// init controller
FOR i:=1 TO 3 DO
	currentRatioMotor2Jnt:=GVL_system_parameters.arm_joint_transmition_efficiency[i-1+Gvl_IO.Joint6]*GVL_system_parameters.arm_joint_torque_constant[i-1+Gvl_IO.Joint6]
							*GVL_system_parameters.transmission_ratio[m_armIdx, i-1+Gvl_IO.Joint6]/1000;
	m_jntPIDCtrl[i].init(GVL_system_parameters.cycle_robot,m_macroJntKp[i],m_macroJntKd[i],m_macroJntKi[i],
		m_macroJntKiLimit[i]* currentRatioMotor2Jnt,	m_macroJnttrlLimit[i]*currentRatioMotor2Jnt);
END_FOR

// init low pass filter
FOR i:=1 TO 3 DO
	m_cmdPosLpf[i].init(i_filterOrd:=1,i_cutoffFreq:=m_jntTargetPosLpfCutoffFreq,i_sampleFreq:=1000);
	m_curJntVelLpf[i].init(i_filterOrd:=1,i_cutoffFreq:=m_curJntVelLpfCutoffFreq,i_sampleFreq:=1000);
END_FOR
END_METHOD

METHOD run : BOOL
VAR_INPUT
	// target joint position in DH model 3
	i_targetJntPos:ARRAY[1..3] OF LREAL;

END_VAR

VAR_OUTPUT
	// motor control current
	o_cmdMotorTrq:ARRAY[1..3] OF LREAL;
END_VAR

VAR
	i: INT;
END_VAR
// fitl target joint position
FOR i:=1 TO 3 DO
	m_targetJntPos[i]:=m_cmdPosLpf[i].run(i_targetJntPos[i]);
END_FOR

// get current joint position
m_curJntPos[1]:=Robot_Status.Robot_Current_DH_Joint_Position_M3[m_armIdx].q1;
m_curJntPos[2]:=Robot_Status.Robot_Current_DH_Joint_Position_M3[m_armIdx].q2;
m_curJntPos[3]:=Robot_Status.Robot_Current_DH_Joint_Position_M3[m_armIdx].q3;

// get current joint velocity
m_curJntVel[1]:=m_curJntVelLpf[1].run(Robot_Status.Robot_Current_Joint_Velocity_V2[m_armIdx,6]);
m_curJntVel[2]:=m_curJntVelLpf[2].run(Robot_Status.Robot_Current_Joint_Velocity_V2[m_armIdx,10]);
m_curJntVel[3]:=m_curJntVelLpf[3].run(Robot_Status.Robot_Current_Joint_Velocity_V2[m_armIdx,11]);

// interpolate command position
FOR i:=1 TO 3 DO
	m_cmdJntVel[i]:=LIMIT(-m_maxJntVel[i],(m_targetJntPos[i]-m_cmdJntPos[i])/GVL_system_parameters.cycle_robot, m_maxJntVel[i]);
	m_cmdJntPos[i]:=m_cmdJntPos[i]+m_cmdJntVel[i]*GVL_system_parameters.cycle_robot;
END_FOR  

// joint position control torque control
FOR i:=1 TO 3 DO
	o_cmdMotorTrq[i]:=0;
	m_posErr[i]:=m_cmdJntPos[i]-m_curJntPos[i];
	m_cmdJntTrq[i]:=m_jntPIDCtrl[i].run(m_cmdJntPos[i],m_curJntPos[i], m_cmdJntVel[i], m_curJntVel[i]);
END_FOR

// safety check
FOR i:=1 TO 3 DO
	IF ABS(m_posErr[i])>m_safetyPosErr[i] THEN
		run := FALSE;
		RETURN;
	END_IF
END_FOR

// motor control current
o_cmdMotorTrq[1]:=gvl_system_parameters.Joint_Motion_direction[m_armIdx,6]*(m_cmdJntTrq[1]+Robot_Status.Robot_Joint_Gravity[1].q6);
o_cmdMotorTrq[2]:=gvl_system_parameters.Joint_Motion_direction[m_armIdx,10]*(m_cmdJntTrq[2]+Robot_Status.Robot_Joint_Gravity[1].q10);
o_cmdMotorTrq[3]:=gvl_system_parameters.Joint_Motion_direction[m_armIdx,11]*(m_cmdJntTrq[3]+Robot_Status.Robot_Joint_Gravity[1].q11);
run := TRUE;
END_METHOD

END_FUNCTION_BLOCK

// ---- FBs_CartControlles/FB_CartPinDeploy.TcPOU
FUNCTION_BLOCK FB_CartPinDeploy EXTENDS FB_CartCtrlBase
VAR_INPUT
END_VAR
VAR_OUTPUT
END_VAR
VAR

	m_actJntPos: Vec8d;
	m_tarJntPos: Vec8d;
	m_initJntPos : Vec8d;
	m_tarJntInc : Vec8d;
	m_maxJntCurrent : ARRAY [1..2] OF LREAL := [1000,1000];
	m_pinDeployed : ARRAY [1..2] OF BOOL; 
	
	m_carJntSoftwareLimit :ARRAY [1..2] OF LREAL := [0.005, 2*g_deg2Rad, 0.005, 2*g_deg2Rad];
	
	// time threshold to 5-8joint after it's enabled
	m_cartAdjustStartWaitTime :LREAL := 0.2;
	
	//adjust start  time 
	m_adjustStartTime :LREAL;

	m_jntOTG :ARRAY [1..2] OF FB_secOrdTrajFilter;
END_VAR

// override this function in each exact controller
METHOD PROTECTED calcCmdJntPos : BOOL
VAR_IN_OUT CONSTANT
	// slave cart joint data
	i_slaveCart :FB_SlaveCart;
END_VAR

VAR
	i:INT;
END_VAR
//In this method, 8 represents the overhang angle
m_adjustStartTime :=LIMIT(0, m_adjustStartTime + g_cartCtrlCycleTime, 1);
m_actJntPos := i_slaveCart.curJntPos;
IF m_adjustStartTime > m_cartAdjustStartWaitTime THEN
	FOR i:=1 TO 2 DO
		IF ABS(i_slaveCart.curJntCurrent[i]) > m_maxJntCurrent[i] THEN
			m_pinDeployed[i] := TRUE;
			m_tarJntPos[i] := m_actJntPos[i];
		END_IF
		
		IF FALSE = m_pinDeployed[i] THEN
			m_tarJntPos[i] := m_actJntPos[i] + GVL_CartControlParameters.g_maxJntVel[i] * g_cartCtrlCycleTime;
		END_IF
		m_jntOTG[i].run(i_targetPos:= m_tarJntPos[i], i_targetVel:= 0.0, o_cmdAcc=> , o_cmdVel=> , o_cmdPos=>m_cmdJntPos[i] );
	END_FOR
	
	IF m_pinDeployed[1] AND m_pinDeployed[2] THEN
		m_isFinished := TRUE;
	END_IF

END_IF
END_METHOD

// override this function in each exact controller
// NOTICE: set joint control mode here, and do some initialization if needed
METHOD PUBLIC init : BOOL
VAR_IN_OUT CONSTANT
	i_slaveCart	:FB_SlaveCart;
END_VAR
VAR_IN_OUT 
	r_cartCtrlCmd :ST_SlaveArmCtrlCmds;
END_VAR
VAR
	i:INT;
END_VAR
//m_holdLastCmds := checkToHoldLastCmds(i_slaveCart);
m_holdLastCmds := checkToHoldLastCmds(i_slaveCart);

SUPER^.init(i_slaveCart,r_cartCtrlCmd);

m_jntEnableFlag[1] :=1;
m_jntEnableFlag[2] :=1;

m_jntOPMode[1]:= DriverOPMode_Pos;
m_jntOPMode[2]:= DriverOPMode_Pos;

m_pinDeployed[1] := FALSE;
m_pinDeployed[2] := FALSE;

m_jntOTG[1].init(i_curCmdPos:= m_cmdJntPos[1], i_curCmdVel:= 0, i_maxV:=GVL_CartControlParameters.g_maxJntVel[1] , i_maxA:=GVL_CartControlParameters.g_maxJntAcc[1] , i_Ts:=g_cartCtrlCycleTime );
m_jntOTG[2].init(i_curCmdPos:= m_cmdJntPos[2], i_curCmdVel:= 0, i_maxV:=GVL_CartControlParameters.g_maxJntVel[2] , i_maxA:=GVL_CartControlParameters.g_maxJntAcc[2] , i_Ts:=g_cartCtrlCycleTime );

m_adjustStartTime := 0;
// update commands to arm
copyCmds(r_cartCtrlCmd);
END_METHOD

END_FUNCTION_BLOCK

// ---- FBs_RobotDynamics/FB_FullArmKinematic.TcPOU
FUNCTION_BLOCK FB_FullArmKinematic
VAR
	m_armIdx :INT :=1;
	
	// nominal DH parameters
	//% setup arm
//% 1        0      0   q1      0
//% 2        90     a2   0      q2
//% 3        -90     0   0       q3
//% 4        0       0   q4      d4
//% 5        -90      0   q5      0

//% paramters definiton:
//% a: distance from joint5 to joint 6 on tool
//% b: distantce form joint 6 to tcp on tool
//% DH definition:
//% index    alpha   a        theta           d
//% 1        90      0        J1+180          0
//% 2        90     42.45     J2-61.935       0
//% P1       0      254       -J2-200.065     0
//% P2       0      305       J2+82              0
//% 3        -90     119.5    0               J3-224.133
//% 4        0       0        J4              -L
//% 5        90      0        J5              0
//% 6        90      a        J6              0
//% tcp      0       b        0               0
	m_armNominalDH :ARRAY[1..14] OF Vec4d;
	
	// calibrated DH parameters err
//	% setupDHErr=[   0   0   dq1     0;
//%                0  da2   0      dq2;
//%                0  0   0       dq3;
//%                0  0   dq4      0;
//%                0  da5  dq5      0];
//% slaveDHErr=[  0       0           dq6      0;
//%               0      0            dq7      da7;
//%               0      0            dq8       0;
//%               0     0               dq9       0;
//%               0     0           0          dq10;
//%                 0       0          0      0];
// m_DHErr=[dq1,da2,dq2, dq3, dq4, da5, dq5,  dq6, dq7, da7, dq8, dq9, dq10]
	m_DHErr:ARRAY[1..13] OF LREAL := [13(0.0)];
	
	// hanger base matrix
	m_baseRadiu :LREAL :=0.17;
	m_baseAng:LREAL := 60.0*g_deg2rad;
	m_baseFrame :ST_Frame;
	
	m_currentDH :ARRAY[1..14] OF Vec4d;
	
	m_tcpFrame :ST_Frame;
	
	m_useCaliData :BOOL:=true;
END_VAR

METHOD init : BOOL
VAR_INPUT
	i_armIdx:INT;
END_VAR
VAR 
	i,j:INT;
END_VAR
m_armIdx := i_armIdx;

FOR i:=1 TO 5 DO 
	FOR j:=1 TO 4 DO
		m_armNominalDH[i][j]:= GVL_SetupArmKinematic.g_setupArmDH[i,j];
	END_FOR	
END_FOR
m_armNominalDH[2][2]:=GVL_SetupArmKinematic.g_setupA2[m_armIdx];
m_armNominalDH[4][4]:=GVL_SetupArmKinematic.g_setupD4[m_armIdx];

FOR i:=1 TO 9 DO 
	FOR j:=1 TO 4 DO
		m_armNominalDH[i+5][j]:= GVL_SlaveArmKinematic.g_slaveArmFullDH[i,j];
	END_FOR	
END_FOR


FOR i:=1 TO 13 DO
	IF m_useCaliData THEN
		m_DHErr[i] := GVL_SlaveArmKinematic.g_slaveArmDHErr[m_armIdx, i];
	ELSE
		m_DHErr[i]:=0;
	END_IF
END_FOR



m_armNominalDH[1][3]:=m_armNominalDH[1][3]+m_DHErr[1];
m_armNominalDH[2][2]:=m_armNominalDH[2][2]+m_DHErr[2];
m_armNominalDH[2][4]:=m_armNominalDH[2][4]+m_DHErr[3];
m_armNominalDH[3][4]:=m_armNominalDH[3][4]+m_DHErr[4];
m_armNominalDH[4][3]:=m_armNominalDH[4][3]+m_DHErr[5];
m_armNominalDH[5][2]:=m_armNominalDH[5][2]+m_DHErr[6];
m_armNominalDH[5][3]:=m_armNominalDH[5][3]+m_DHErr[7];

m_armNominalDH[6][3]:=m_armNominalDH[6][3]+m_DHErr[8];
m_armNominalDH[7][3]:=m_armNominalDH[7][3]+m_DHErr[9];
m_armNominalDH[7][4]:=m_armNominalDH[7][4]+m_DHErr[10];
m_armNominalDH[8][3]:=m_armNominalDH[8][3]+m_DHErr[11];
m_armNominalDH[9][3]:=m_armNominalDH[9][3]+m_DHErr[12];
m_armNominalDH[10][4]:=m_armNominalDH[10][4]+m_DHErr[13];

m_baseFrame.m_pos[3]:=0;
IF (m_armIdx=1) THEN
	m_baseFrame.m_pos[1]:=-m_baseRadiu; 
	m_baseFrame.m_pos[2]:=0;
	
ELSIF (m_armIdx=2) THEN
	m_baseFrame.m_pos[1]:=-m_baseRadiu*COS(m_baseAng); 
	m_baseFrame.m_pos[2]:=-m_baseRadiu*SIN(m_baseAng);
	
ELSIF (m_armIdx=3) THEN	
	m_baseFrame.m_pos[1]:=m_baseRadiu*COS(m_baseAng); 
	m_baseFrame.m_pos[2]:=-m_baseRadiu*SIN(m_baseAng); 
	
ELSIF (m_armIdx=4) THEN	
	m_baseFrame.m_pos[1]:=m_baseRadiu; 
	m_baseFrame.m_pos[2]:=0;
END_IF

IF m_useCaliData THEN
	m_baseFrame.m_pos[1]:=m_baseFrame.m_pos[1]+GVL_SlaveArmKinematic.g_slaveArmBaseErr[m_armIdx,1];
	m_baseFrame.m_pos[2]:=m_baseFrame.m_pos[2]+GVL_SlaveArmKinematic.g_slaveArmBaseErr[m_armIdx,2];
END_IF
m_baseFrame.m_rot[1,1]:=0;
m_baseFrame.m_rot[2,1]:=1;
m_baseFrame.m_rot[3,1]:=0;

m_baseFrame.m_rot[1,2]:=-1;
m_baseFrame.m_rot[2,2]:=0;
m_baseFrame.m_rot[3,2]:=0;

m_baseFrame.m_rot[1,3]:=0;
m_baseFrame.m_rot[2,3]:=0;
m_baseFrame.m_rot[3,3]:=1;
END_METHOD

METHOD run : BOOL
VAR_IN_OUT CONSTANT
	// setup joint angle
	i_setupPos : vec5d;
	
	// slave DH joint angle
	i_slaveDHJntPos :Vec6d;
	
	// instrument
	i_instruStatus :ST_InstruStatus;
END_VAR
VAR_IN_OUT
	r_tcpPose:ST_Frame;
END_VAR
VAR
	i:INT;
	T1,T2 :ST_Frame;
END_VAR
// instrument parameters
m_armNominalDH[11][4]:=-GVL_SlaveArmKinematic.g_L;
m_armNominalDH[13][2]:=GVL_SlaveArmKinematic.g_a;
m_armNominalDH[14][2]:=GVL_SlaveArmKinematic.g_b;
FOR i:=1 TO g_instruTypeNum DO 
	IF g_instruTypePool[i].m_InstruID = i_instruStatus.m_type THEN
		m_armNominalDH[11][4]:=-(g_instruTypePool[i].m_rodLength-GVL_SlaveArmKinematic.g_panelHeight);
		m_armNominalDH[13][2]:=g_instruTypePool[i].m_headLength;
		m_armNominalDH[14][2]:=g_instruTypePool[i].m_fingerLength;
		EXIT;
	END_IF
END_FOR

// add joint position
m_currentDH:=m_armNominalDH;
m_currentDH[1][3]:=m_currentDH[1][3]+i_setupPos[1];
m_currentDH[2][4]:=m_currentDH[2][4]+i_setupPos[2];
m_currentDH[3][4]:=m_currentDH[3][4]+i_setupPos[3];
m_currentDH[4][3]:=m_currentDH[4][3]+i_setupPos[4];
m_currentDH[5][3]:=m_currentDH[5][3]+i_setupPos[5];
m_currentDH[6][3]:=m_currentDH[6][3]+i_slaveDHJntPos[1];
m_currentDH[7][3]:=m_currentDH[7][3]+i_slaveDHJntPos[2];
m_currentDH[8][3]:=m_currentDH[8][3]-i_slaveDHJntPos[2];
m_currentDH[9][3]:=m_currentDH[9][3]+i_slaveDHJntPos[2];
m_currentDH[10][4]:=m_currentDH[10][4]+i_slaveDHJntPos[3];
m_currentDH[11][3]:=m_currentDH[11][3]+i_slaveDHJntPos[4];
m_currentDH[12][3]:=m_currentDH[12][3]+i_slaveDHJntPos[5];
m_currentDH[13][3]:=m_currentDH[13][3]+i_slaveDHJntPos[6];

m_tcpFrame:= m_baseFrame;
FOR i:=1 TO 14 DO 
	T1:=DHTrans(m_currentDH[i]);
	T2:=transform(m_tcpFrame,T1);
	m_tcpFrame:=T2;
END_FOR
matMultiply(T2.m_rot, GVL_SlaveArmKinematic.g_tcpRotation, m_tcpFrame.m_rot);

r_tcpPose:=m_tcpFrame;
END_METHOD

END_FUNCTION_BLOCK

// ---- FBs_RobotDynamics/FB_InstruViewCheck.TcPOU
FUNCTION_BLOCK FB_InstruViewCheck
VAR
	
	// scoep projection matrix 
	//SN: HA21938730
	m_scopeRot :Mat3d :=[0.9983, -0.0327, 0.048, 
						0.0319, 0.9993, 0.0179,
						-0.0486, -0.0164, 0.9987];
	m_scopePos :Vec3d:= [0.005, 0.000214, 0.00386];
	m_scopeFocal :LREAL :=1400;
	
//	//SN: HA20160831
//	m_scopeRot :Mat3d :=[0.9952, 0.0185, 0.0961, 
//						-0.0177, 0.9998, -0.0099,
//						-0.0963, 0.0081, 0.9953];
//	m_scopePos :Vec3d:= [-0.0006967, 0.001848, -0.005];
//	m_scopeFocal :LREAL :=1420;

	// arm kinematic function block
	m_armKinematic :ARRAY[1..g_sArmNum] OF FB_FullArmKinematic;
	
	// instrument pose
	m_instruReady:ARRAY[1..g_sArmNum] OF BOOL;
	m_instruPose :ARRAY[1..g_sArmNum] OF ST_Frame;
	
	// endoscope pose
	m_scopeReady :BOOL;
	m_scopePose : ST_Frame;
	
	// instrument pose in scope 
	m_instruPoseInScope :ARRAY[1..g_sArmNum] OF ST_Frame;
	
	// instrument position in image([x_pixel, y_pixel, z_dir])
	m_instruImgPos :ARRAY[1..g_sArmNum] OF Vec3d;
	
	// out-view instrument position on image boundary([x_pixel, y_pixel, z_dir])
	 m_instruImgBoundPos :ARRAY[1..g_sArmNum] OF Vec3i;
	 
	 // image boundary
	 m_imgWidth :INT := 960;
	 m_ImgHeight :INT :=540;
	
END_VAR

METHOD init : BOOL
VAR_INPUT
END_VAR
VAR
	i:INT;
END_VAR
FOR i:=1 TO g_sArmNum DO
	m_instruReady[i]:=FALSE;
	m_armKinematic[i].init(i);
	m_instruImgPos[i]:=g_zeroVec3d;
	m_instruImgBoundPos[i]:=g_zeroVec3i;
END_FOR
m_scopeReady:=FALSE;
END_METHOD

METHOD run : BOOL
VAR_IN_OUT CONSTANT
	// setup joint position
	i_setupJntPos :ARRAY[1..g_sArmNum] OF Vec5d;
	
	// slave joint position
	i_slaveDHJntPos :ARRAY[1..g_sArmNum] OF Vec6d;
	
	// instrument info
	i_instruInfo : ARRAY[1..g_sArmNum] OF ST_InstruStatus;
END_VAR

VAR
	i:INT;
	tmpFrame: ST_Frame;
	newPos:Vec3d ;
	xb,yb : INT;
END_VAR
m_scopeReady := FALSE;
// update instrument and endoscope pose
FOR i:=1 TO g_sArmNum DO 
	m_instruReady[i]:=FALSE;
	IF i_instruInfo[i].m_ready THEN
		m_instruReady[i]:=TRUE;
		m_armKinematic[i].run(i_setupJntPos[i],i_slaveDHJntPos[i], i_instruInfo[i], m_instruPose[i]);
		IF i_instruInfo[i].m_type = InstruType_Endoscope THEN
			m_scopePose := m_instruPose[i];
			m_scopeReady := TRUE;
		END_IF
	END_IF
	
	m_instruImgPos[i]:=g_zeroVec3d;
	m_instruImgBoundPos[i]:=g_zeroVec3i;
END_FOR

IF m_scopeReady THEN
	FOR i:=1 TO g_sArmNum DO
		IF m_instruReady[i] THEN
			// calculate instrument pose in endoscope
			tmpFrame :=invFrame(m_scopePose);
			m_instruPoseInScope[i] := transform(tmpFrame, m_instruPose[i]);
			
			// calculate instrument in image
			IF ABS(m_instruPoseInScope[i].m_pos[3])>0.02 THEN
				MatMultiVec(m_scopeRot, m_instruPoseInScope[i].m_pos, newPos);
				vecSelfAdd(newPos, m_scopePos);
				m_instruImgPos[i][1]:= m_scopeFocal* newPos[1]/ABS(newPos[3]);
				m_instruImgPos[i][2]:= -m_scopeFocal * newPos[2]/ABS(newPos[3]);
				m_instruImgPos[i][3] := sign(newPos[3]); 
			END_IF
			
			// check if instrument is  out of view
			IF ABS(m_instruImgPos[i][1])>m_imgWidth OR ABS(m_instruImgPos[i][2])>m_ImgHeight THEN
				IF ABS(m_instruImgPos[i][2]/m_instruImgPos[i][1]) > INT_TO_LREAL( m_ImgHeight)/INT_TO_LREAL(m_imgWidth) THEN
					yb:=sign(m_instruImgPos[i][2])*m_ImgHeight;
					xb:=LREAL_TO_INT(m_instruImgPos[i][1]*yb/m_instruImgPos[i][2]);
				ELSE
					xb:=sign(m_instruImgPos[i][1])*m_imgWidth;
					yb:=LREAL_TO_INT(m_instruImgPos[i][2]*xb/m_instruImgPos[i][1]);
				END_IF
				m_instruImgBoundPos[i][1]:=xb;
				m_instruImgBoundPos[i][2]:=yb;
				m_instruImgBoundPos[i][3]:=LREAL_TO_INT(m_instruImgPos[i][3]);
			END_IF
						
		END_IF
	END_FOR
END_IF
END_METHOD

END_FUNCTION_BLOCK

// ---- FBs_RobotDynamics/FB_SlaveDynamic.TcPOU
FUNCTION_BLOCK FB_SlaveDynamic
VAR_INPUT
END_VAR
VAR_OUTPUT
END_VAR
VAR CONSTANT
	//kinematic constraint
	//  q3 =- q2;           
	//  q4 = q2;             
 	// jacobian with active joints
 	// jaco_DH*qdot_DH = jaco_DH * (A * qdot_active)= jaco * qdot_active
 	// q_DH=[q1,q2,q3,q4,q5];
 	// q_active=[q1,q2,q5]
	m_jacoA :Mat53 :=
	[   1,  0,  0,
        0,  1,  0,
		0, -1,  0,
		0,  1,  0,
		0,  0,  1];
	
	// DH parameters for dynamic model
	(*slaveDH=[   deg90       0           q1+pi                502.591/1000;
            deg90       42.45/1000  q2-deg2rad(61.935)   0;
            0           254/1000    q3-deg2rad(200.065) 0;
            0           305/1000    q4+deg2rad(82)       0;
            -deg90      119.5/1000  0                           q5-224.133/1000];*)
	m_armOriginalDH:ARRAY[1..5,1..4] OF LREAL :=
	[PI/2,       0,         	   pi,     502.591/1000,          
	PI/2,       42.45/1000,  	-61.935*g_deg2rad,  0, 		
	0,           254.0/1000,  	-200.065*g_deg2rad, 0,  
	0,           305.0/1000,    	82*g_deg2rad,      	0, 			
	-PI/2,      119.5/1000,   0,	-224.133/1000];
	
END_VAR

VAR
			
	m_armIdx :INT;
	m_armDH:ARRAY[1..5] OF Vec4d;
	
	// dynamic parameters
	m_linkMass :ARRAY[1..5] OF LREAL;
	m_linkCOM :ARRAY[1..5] OF Vec3d;
	m_linkInertia :ARRAY[1..5] OF Mat3d;
		
	// frame of each joint
	m_jntFrame :ARRAY[1..5] OF ST_Frame;
	
	// jacobian of mass center
	m_Jp :ARRAY[1..5] OF Mat3d;
	m_Jo :ARRAY[1..5] OF Mat3d;
	
	// motor inertia at link size
	m_motorInertia :Vec3d;
	
	// mass matrix in joint space
	m_massMat :Mat3d;
	
END_VAR

METHOD init : BOOL
VAR_INPUT
	i_armIdx :INT ;
END_VAR

VAR
	i,j:INT;
END_VAR
m_armIdx:=i_armIdx;

m_linkMass:=GVL_SlaveArmDynamics.g_linkMass;
FOR i:=1 TO 5 DO
	m_linkCOM[i][1]:=GVL_SlaveArmDynamics.g_linkCOM[i,1];
	m_linkCOM[i][2]:=GVL_SlaveArmDynamics.g_linkCOM[i,2];
	m_linkCOM[i][3]:=GVL_SlaveArmDynamics.g_linkCOM[i,3];
	
	m_linkInertia[i][1,1]:=GVL_SlaveArmDynamics.g_linkInertia[i,1];
	m_linkInertia[i][2,2]:=GVL_SlaveArmDynamics.g_linkInertia[i,2];
	m_linkInertia[i][3,3]:=GVL_SlaveArmDynamics.g_linkInertia[i,3];
	m_linkInertia[i][1,2]:=GVL_SlaveArmDynamics.g_linkInertia[i,4];
	m_linkInertia[i][1,3]:=GVL_SlaveArmDynamics.g_linkInertia[i,5];
	m_linkInertia[i][2,3]:=GVL_SlaveArmDynamics.g_linkInertia[i,6];
	m_linkInertia[i][2,1]:=m_linkInertia[i][1,2];
	m_linkInertia[i][3,1]:=m_linkInertia[i][1,3];
	m_linkInertia[i][3,2]:=m_linkInertia[i][2,3];
END_FOR

FOR i:=1 TO 3 DO
	m_motorInertia[i]:=GVL_SlaveArmDynamics.g_motorInertia[i]*GVL_SlaveMotorParameters.g_motorReduction[i]*GVL_SlaveMotorParameters.g_motorReduction[i];
END_FOR

FOR i:=1 TO 5 DO
	FOR j:=1 TO 4 DO 
		m_armDH[i][j] := m_armOriginalDH[i,j];
	END_FOR
END_FOR
END_METHOD

PROPERTY PUBLIC jntMassMat : Mat3d
GET
jntMassMat := m_massMat;
END_GET
END_PROPERTY

// update dynamic and kinematic data 
METHOD updateDynamic : BOOL
VAR_IN_OUT CONSTANT
	i_jntPos : Vec8d;
END_VAR
VAR
	tmpJntPos :Vec8d;
	
	i,j:INT;
	m,n :INT;
	linkMassMat :ARRAY[1..5] OF Mat3d;
	linkInerMat :ARRAY[1..5] OF Mat3d;
	inertia,Rt :Mat3d;
	
	JotI,Jot, Jpt :Mat3d;
	
	tmpMat3d :Mat3d;

	
END_VAR
// update kinematic 
updateKinematic(i_jntPos);

// joint space mass matrix
// massMat=m*Jp'*Jp+Jo'*R*I*R'*Jo
FOR i:=1 TO 5 DO
	// iner=R*I*R'
	matMultiply(m_jntFrame[i].m_rot,m_linkInertia[i],tmpMat3d);
	matTranspose(m_jntFrame[i].m_rot, Rt);
	matMultiply(tmpMat3d,Rt,inertia);
	
	// m*Jp'*Jp+Jo'*iner*Jo
	matTranspose(m_Jp[i],Jpt);
	matMultiply(Jpt,m_Jp[i], tmpMat3d);
	matMultiNum(tmpMat3d, m_linkMass[i],linkMassMat[i]);
	
	matTranspose(m_Jo[i],Jot);
	matMultiply(Jot,inertia, JotI);
	matMultiply(JotI,m_Jo[i],linkInerMat[i]);
END_FOR

// total mass mat
m_massMat :=g_zeroMat3d;
FOR i:=1 TO 5 DO
	matSelfAdd(m_massMat,linkMassMat[i]);
	matSelfAdd(m_massMat,linkInerMat[i]);
END_FOR

// add motor inertial 
FOR i:=1 TO 3 DO
	m_massMat[i,i]:=m_massMat[i,i]+m_motorInertia[i];
END_FOR
END_METHOD

// only update kinematic data
METHOD PROTECTED updateKinematic : BOOL
VAR_IN_OUT CONSTANT
	i_jntPos : Vec8d;
END_VAR
VAR
	Jp :Mat35;
	Jo :Mat35;
	T :ST_Frame;
	i,j:INT;
	Pc,z,p:Vec3d;
	m,n :INT;
	
END_VAR
// tranform a joint positon to DH ones
m_armDH[1][3] := m_armOriginalDH[1,3] + i_jntPos[1];
m_armDH[2][3] := m_armOriginalDH[2,3] + i_jntPos[2];
m_armDH[3][3] := m_armOriginalDH[3,3] - i_jntPos[2];
m_armDH[4][3] := m_armOriginalDH[4,3] + i_jntPos[2];
m_armDH[5][4] := m_armOriginalDH[5,4] + i_jntPos[3];

// compute joint frame
m_jntFrame[1]:=DHTrans(m_armDH[1]);
T:=DHTrans(m_armDH[2]);
m_jntFrame[2]:=transform(m_jntFrame[1],T);
T:=DHTrans(m_armDH[3]);
m_jntFrame[3]:=transform(m_jntFrame[2],T);
T:=DHTrans(m_armDH[4]);
m_jntFrame[4]:=transform(m_jntFrame[3],T);
T:=DHTrans(m_armDH[5]);
m_jntFrame[5]:=transform(m_jntFrame[4],T);


// jacobian of mass center
FOR i:=1 TO 5 DO 
	Jp := g_zeroMat35;
	Jo := g_zeroMat35;
    T:=m_jntFrame[i];
	// mass center world position
    matMultiVec(T.m_rot,m_linkCOM[i], Pc);
	vecSelfAdd(Pc, T.m_pos);
    FOR j:=1 TO i DO
        T:=m_jntFrame[j];
		z[1]:=T.m_rot[1,3];
		z[2]:=T.m_rot[2,3];
		z[3]:=T.m_rot[3,3];
		IF (5=j) THEN
			Jp[1,j]:=z[1];
			Jp[2,j]:=z[2];
			Jp[3,j]:=z[3];
			Jo[1,j]:=0;
			Jo[2,j]:=0;
			Jo[3,j]:=0;
		ELSE
			vecSub(Pc,T.m_pos,p);
			p:=cross(z,p);
			Jp[1,j]:=p[1];
			Jp[2,j]:=p[2];
			Jp[3,j]:=p[3];
			Jo[1,j]:=z[1];
			Jo[2,j]:=z[2];
			Jo[3,j]:=z[3];			
        END_IF
    END_FOR
	// multiply m_jacoA
	matMultiply(Jp, m_jacoA, m_Jp[i]);
	matMultiply(Jo, m_jacoA, m_Jo[i]);
END_FOR
END_METHOD

END_FUNCTION_BLOCK

// ---- FBs_RobotDynamics/FB_SlaveGravity.TcPOU
FUNCTION_BLOCK FB_SlaveGravity
VAR_INPUT
END_VAR
VAR
	m_armIdx :INT ;

	// current arm parameters
	m_armParams :ARRAY[1..5] OF LREAL;

END_VAR

METHOD getRegMat : BOOL
VAR_INPUT
	// joint position of setup joint, joint6-8
	setupAng :LREAL;
	q1: LREAL;
	q2: LREAL;
	q3: LREAL;
END_VAR

VAR
	s0,c0, s1,c1,s2, c2,d3 :LREAL;
END_VAR

VAR_OUTPUT
	o_regMat:ARRAY[1..3,1..5] OF LREAL;
END_VAR
s0:=SIN(setupAng);
c0:=COS(setupAng);
s1:=SIN(q1);
c1:=COS(q1);
s2:=SIN(q2);
c2:=COS(q2);
d3:=q3;

// joint1
o_regMat[1,1] :=s0*s1*s2*d3;
o_regMat[1,2] :=  s0*s1;
o_regMat[1,3] := -s0*c1;
o_regMat[1,4] := s0*s1*s2;
o_regMat[1,5] := s0*c2*s1 ;

// joint2 
o_regMat[2,1] :=  - (c0*s2*d3+s0*c1*c2*d3);
o_regMat[2,2] := 0;
o_regMat[2,3] := 0;
o_regMat[2,4] :=  - (c0*s2+s0*c1*c2);
o_regMat[2,5] := s0*c1*s2- c0*c2;

// joint3
o_regMat[3,1] :=c0*c2 - s0*c1*s2;
o_regMat[3,2] :=0;
o_regMat[3,3] :=0;
o_regMat[3,4] :=0;
o_regMat[3,5] :=0;
END_METHOD

METHOD init : BOOL
VAR_INPUT
	i_armIdx :INT;
END_VAR
m_armIdx :=i_armIdx;
END_METHOD

METHOD run : Vec3d
VAR_IN_OUT CONSTANT
	// setup joint5 angle
	i_setupPos :LREAL;
	
	// slave joint angle
	i_slaveJntPos :Vec8d;
	
	// instrument
	i_instruStatus :ST_InstruStatus;
END_VAR
VAR
	q1, q2, q3 :LREAL;
	i,j:INT;
	
	// gravity regression matrix
	regMat:ARRAY[1..3,1..5] OF LREAL;
END_VAR
q1 :=LIMIT (GVL_SlaveMotorParameters.g_minJntPos[1], i_slaveJntPos[1], GVL_SlaveMotorParameters.g_maxJntPos[1]);
q2 := LIMIT (GVL_SlaveMotorParameters.g_minJntPos[2], i_slaveJntPos[2], GVL_SlaveMotorParameters.g_maxJntPos[2]);
q3 := LIMIT (GVL_SlaveMotorParameters.g_minJntPos[3], i_slaveJntPos[3], GVL_SlaveMotorParameters.g_maxJntPos[3]);


// get regression matrx
getRegMat(i_setupPos, q1, q2, q3, o_regMat=>regMat);

// determine current arm parameters
IF FALSE = i_instruStatus.m_ready THEN
	// arm only
	FOR i:=1 TO 5 DO
		m_armParams[i]:=GVL_SlaveArmDynamics.g_gravityParam[m_armIdx,i];
	END_FOR

// endoscope
ELSIF InstruType_endoscope = i_instruStatus.m_type THEN 
	FOR i:=1 TO 5 DO
		m_armParams[i]:=GVL_SlaveArmDynamics.g_gravityParam[m_armIdx,i]+GVL_SlaveArmDynamics.g_gravityEndoscope[i];
	END_FOR

// instrument
ELSE
	FOR i:=1 TO 5 DO
		m_armParams[i]:=GVL_SlaveArmDynamics.g_gravityParam[m_armIdx,i]+GVL_SlaveArmDynamics.g_gravityInstrument[i];
	END_FOR
// TODO:Trocar
END_IF

// calculate gravity torque
FOR i:=1 TO 3 DO
	run[i]:=0;
	FOR j:=1 TO 5 DO
		run[i]:=run[i]+regMat[i,j]*m_armParams[j];
	END_FOR
END_FOR
END_METHOD

END_FUNCTION_BLOCK

// ---- FBs_RobotDynamics/FB_SetupGravity.TcPOU
FUNCTION_BLOCK FB_SetupGravity
VAR_INPUT
END_VAR
VAR
	m_armIdx :INT ;

	// current arm parameters
	m_armParams :ARRAY[1..7] OF LREAL;

	// gravity regression matrix
	regMat:ARRAY[1..7] OF LREAL;
	
	m_graivty :LREAL;
END_VAR

METHOD getRegMat : BOOL
VAR_INPUT
	// joint position of setup joint, joint6-8
	setupAng :LREAL;
	q1: LREAL;
	q2: LREAL;
	q3: LREAL;
END_VAR

VAR
	s0,c0,s1,c1,s2, c2,d3 :LREAL;
END_VAR

VAR_OUTPUT
	o_regMat:ARRAY[1..7] OF LREAL;
END_VAR
s0:= SIN(setUpAng);
c0:= COS(setUpAng);
s1:=SIN(q1);
c1:=COS(q1);
s2:=SIN(q2);
c2:=COS(q2);
d3:=q3;

// setup joint
o_regMat[1] :=c0;
o_regMat[2] := s0;
o_regMat[3] :=-(c2*s0*d3+c0*c1*s2*d3);
o_regMat[4] :=  -c0*c1;
o_regMat[5] :=  -c0*s1;
o_regMat[6] := - (c0*c1*s2+c2*s0);
o_regMat[7] :=  s0*s2- c0*c1*c2  ;
END_METHOD

METHOD init : BOOL
VAR_INPUT
	i_armIdx :INT;
END_VAR
m_armIdx :=i_armIdx;
END_METHOD

METHOD run : BOOL
VAR_IN_OUT CONSTANT
	// setup joint angle
	i_setupJntPos :Vec5d;
	
	// slave joint angle
	i_slaveJntPos :Vec8d;
	
	// instrument
	i_instruStatus :ST_InstruStatus;
END_VAR
VAR_OUTPUT
	// setup joint3 gravity
	o_jnt3Gravity :LREAL;
	
	// setup joint5 gravity
	o_jnt5Gravity :LREAL;
END_VAR
VAR
	setupPos, q1, q2, q3 :LREAL;
	i,j:INT;
	
	gravityTrq :Vec4d;

END_VAR
setupPos:=LIMIT(GVL_SetupMotorParameters.g_minJntPos[m_armIdx,5], i_setupJntPos[5], GVL_SetupMotorParameters.g_maxJntPos[m_armIdx,5]);
q1 :=LIMIT (GVL_SlaveMotorParameters.g_minJntPos[1], i_slaveJntPos[1], GVL_SlaveMotorParameters.g_maxJntPos[1]);
q2 := LIMIT (GVL_SlaveMotorParameters.g_minJntPos[2], i_slaveJntPos[2], GVL_SlaveMotorParameters.g_maxJntPos[2]);
q3 := LIMIT (GVL_SlaveMotorParameters.g_minJntPos[3], i_slaveJntPos[3], GVL_SlaveMotorParameters.g_maxJntPos[3]);

// get regression matrx
getRegMat(setupPos, q1, q2, q3, o_regMat=>regMat);

// determine current arm parameters
m_armParams[1] := GVL_SetupArmDynamics.g_setupJnt5GravityParam[m_armIdx,1];
m_armParams[2] := GVL_SetupArmDynamics.g_setupJnt5GravityParam[m_armIdx,2];
IF FALSE = i_instruStatus.m_ready THEN
	// arm only
	FOR i:=1 TO 5 DO
		m_armParams[i+2]:= GVL_SlaveArmDynamics.g_gravityParam[m_armIdx,i];
	END_FOR

// endoscope
ELSIF InstruType_endoscope = i_instruStatus.m_type THEN 
	FOR i:=1 TO 5 DO
		m_armParams[i+2]:=GVL_SlaveArmDynamics.g_gravityParam[m_armIdx,i]+GVL_SlaveArmDynamics.g_gravityEndoscope[i];
	END_FOR

// instrument
ELSE
	FOR i:=1 TO 5 DO
		m_armParams[i+2]:=GVL_SlaveArmDynamics.g_gravityParam[m_armIdx,i]+GVL_SlaveArmDynamics.g_gravityInstrument[i];
	END_FOR
// TODO:Trocar
END_IF

// calculate gravity torque
o_jnt5Gravity:=0;
FOR j:=1 TO 7 DO
	o_jnt5Gravity:=o_jnt5Gravity+regMat[j]*m_armParams[j];
END_FOR
m_graivty := o_jnt5Gravity;

o_jnt3Gravity:= setupJnt3Gravity(i_setupJntPos[3]);
END_METHOD

METHOD setupJnt3Gravity : LREAL
VAR_INPUT
	i_jnt3Pos :LREAL;
END_VAR
VAR
	q:LREAL;
END_VAR
q := LIMIT(GVL_SetupArmDynamics.g_setupJnt3GravityPosRange[m_armIdx,1], i_jnt3Pos, GVL_SetupArmDynamics.g_setupJnt3GravityPosRange[m_armIdx,2]);
setupJnt3Gravity:=GVL_SetupArmDynamics.g_setupJnt3GravityParams[m_armIdx,1]*EXPT(q,3)+GVL_SetupArmDynamics.g_setupJnt3GravityParams[m_armIdx,2]*EXPT(q,2)+
				GVL_SetupArmDynamics.g_setupJnt3GravityParams[m_armIdx,3]*q+GVL_SetupArmDynamics.g_setupJnt3GravityParams[m_armIdx,4];
END_METHOD

END_FUNCTION_BLOCK

// ---- FBs_Robots/FB_SetupArm.TcPOU
FUNCTION_BLOCK FB_SetupArm
VAR_INPUT
END_VAR
VAR_OUTPUT
END_VAR
VAR
	// arm index, from 1 to 4
	m_armIdx: INT;
	
	// joints
	m_joints :ARRAY[1..g_setupJntNum] OF FB_SetupJoint;
	
	// adjust detect
	m_adjustIO AT%I* :UDINT;
	m_manualAdjustOnFlag :BOOL;
	m_jnt5AdjustDir :INT; // -1, 0, 1;
	m_manualAdjustDetect : FB_setupAdjustDetect;
	m_jnt5AdjustDetect : FB_setupJnt5AdjustDetect;
	
	// arm cartesian data, defined in cart origin
	m_curCartPose	:ST_Frame;
	
	// cartesion position of remote center
	m_rcPos :Vec3d;	
	
	// arm joint data
	m_curMotorPos :Vec5d;
	m_curLinkPos :Vec5d;
	m_curJntPos :Vec5d;
	m_curJntVel :Vec5d;
	m_curJntTrq :Vec5d;
	m_rawJntCurrent :Vec5d;
	m_filtJntCurrent :Vec5d;
	m_cmdJntCurrent : Vec5d;
	m_cmdJntPos :Vec5d;
	m_cmdJntVel :Vec5d;
	m_cmdJntTrq :Vec5d;
		
	// arm gravity
	m_jntGravity : Vec5d:=g_zeroVec5d;
	
	// joint position controller
	m_jntPIDCtrl :ARRAY[1..g_setupJntNum] OF FB_PID;
	
	//arm light out to drive
	m_lightIO AT %Q* :DINT;
	
	// output arm light
	m_SdoWrite:ARRAY [1..2] OF FB_EcCoESdoWrite;
	
	//IP of operating arm
	m_armNetId:T_AmsNetId; 	
	
	//Joint port number
	m_jointAddrJ8:UINT;	
	m_jointAddrPbox:UINT;
	
END_VAR

PROPERTY armIdx : int
GET
armIdx:=m_armIdx;
END_GET
END_PROPERTY

METHOD PROTECTED checkIO : BOOL
VAR_INPUT
END_VAR
// check manual and auto adjust button
m_manualAdjustOnFlag := m_manualAdjustDetect.run(m_adjustIO);
m_jnt5AdjustDir := m_jnt5AdjustDetect.run(m_adjustIO);
END_METHOD

METHOD checkLight : BOOL
VAR_INPUT
	i_lightCtrlWord : UDINT;
END_VAR

VAR
	lightCtrlWord : UDINT;
END_VAR
// to PDO
m_lightIO := UDINT_TO_DINT(i_lightCtrlWord);

// trig sdo write
lightCtrlWord := SHL(i_lightCtrlWord,16);
m_SdoWrite[1](sNetId:= m_armNetId, nSlaveAddr:= m_jointAddrJ8, nSubIndex:= 0, nIndex:= 16#6097, pSrcBuf:=ADR(lightCtrlWord) , cbBufLen:=SIZEOF(lightCtrlWord) , bExecute:= TRUE, tTimeout:= , bBusy=> , bError=> , nErrId=> );
m_SdoWrite[2](sNetId:= m_armNetId, nSlaveAddr:= m_jointAddrPbox, nSubIndex:= 0, nIndex:= 16#6097, pSrcBuf:= ADR(lightCtrlWord), cbBufLen:= SIZEOF(lightCtrlWord), bExecute:= TRUE, tTimeout:= , bBusy=> , bError=> , nErrId=> );

// disable sdo write
IF NOT m_SdoWrite[1].bBusy AND  NOT m_SdoWrite[2].bBusy THEN
	m_SdoWrite[1](bExecute:=FALSE);
	m_SdoWrite[2](bExecute:=FALSE);
END_IF
END_METHOD

PROPERTY cmdJntCurrent : REFERENCE TO  Vec5d
GET
cmdJntCurrent ref= m_cmdJntCurrent;
END_GET
END_PROPERTY

PROPERTY curCartPose : REFERENCE TO ST_Frame
GET
curCartPose ref=m_curCartPose;
END_GET
END_PROPERTY

PROPERTY curJntPos : REFERENCE TO Vec5d
GET
curJntPos ref=m_curJntPos;
END_GET
END_PROPERTY

PROPERTY curJntTrq : REFERENCE TO Vec5d
GET
curJntTrq ref=m_curJntTrq;
END_GET
END_PROPERTY

PROPERTY curJntVel :REFERENCE TO Vec5d
GET
curJntVel ref=m_curJntVel;
END_GET
END_PROPERTY

PROPERTY curLinkPos :REFERENCE TO Vec5d
GET
curLinkPos ref=m_curLinkPos;
END_GET
END_PROPERTY

PROPERTY curMotorPos : REFERENCE TO  Vec5d
GET
curMotorPos ref=m_curMotorPos;
END_GET
END_PROPERTY

METHOD PUBLIC enable : BOOL
VAR_IN_OUT CONSTANT
	i_jntIdx :Vec5i;
END_VAR
VAR
	i :INT ;
END_VAR
FOR i:=1 TO g_setupJntNum DO
	IF 1= i_jntIdx[i] THEN
		m_joints[i].enable();
	ELSE
		m_joints[i].disable();
	END_IF
END_FOR
END_METHOD

PROPERTY filtJntCurrent :REFERENCE TO Vec5d
GET
filtJntCurrent ref= m_filtJntCurrent;
END_GET
END_PROPERTY

// compute cartesion pose in cart origin
METHOD PROTECTED forwardKinematic : BOOL
VAR_IN_OUT CONSTANT
	i_jntPos :Vec5d;
END_VAR
VAR_IN_OUT
	r_cartPose :ST_Frame;
	
	// position of remote center
	r_rcPos :Vec3d;
END_VAR
VAR
	a2,d4,d6:LREAL; //DH parameters
	
	Radius,Angle,R1,q:LREAL; //Disk structure parameters
	x,y,z:LREAL;
	basePosMatrix:ARRAY[1..4,1..4] OF LREAL;//transform from origin to C0
	
	T_50:ARRAY[1..4,1..4] OF LREAL; //transform from C0 to C5
	F5:ARRAY[1..4,1..4] OF LREAL; //transform from origin to C5
	q1,q2,q3,q4,q5:LREAL;	
	c14,s14,c5,s5,s1,c1:LREAL;
	
	fixPointTransform:ARRAY[1..4,1..4] OF LREAL; //transform from C5 to fixed point
	fixPointMatrix:ARRAY[1..4,1..4] OF LREAL;
END_VAR
//TODO: move DH parameter to GVL 


//****************input:five joint position of SetupArm********************//
q1:=i_jntPos[1]; q2:=i_jntPos[2]; q3:=i_jntPos[3]; q4:=i_jntPos[4]; q5:=i_jntPos[5];

//**********************DH parameters*************************//
IF (m_armIdx=1) THEN
	a2:=0.019; d4:=0.5205;
	
ELSIF (m_armIdx=2) THEN
	a2:=0.136; d4:=0.3545;
	
ELSIF (m_armIdx=3) THEN	
	a2:=0.136; d4:=0.3545;
	
ELSIF (m_armIdx=4) THEN	
	a2:=0.1825; d4:=0.5205;
END_IF
d6:=0.6387229+0.1659;

//********************transform form origin to C0***********************//
Radius:=0.170; Angle:=60.0*g_deg2Rad;
R1:=Radius;  q:=Angle;
IF (m_armIdx=1) THEN
	x:=-R1; y:=0; z:=0;
	
ELSIF (m_armIdx=2) THEN
	x:=-R1*COS(q); y:=-R1*SIN(q); z:=0;
	
ELSIF (m_armIdx=3) THEN	
	x:=R1*COS(q); y:=-R1*SIN(q); z:=0;
	
ELSIF (m_armIdx=4) THEN	
	x:=R1; y:=0; z:=0;
END_IF

basePosMatrix[1,1]:=0;
basePosMatrix[2,1]:=1;
basePosMatrix[3,1]:=0;
basePosMatrix[4,1]:=0;

basePosMatrix[1,2]:=-1;
basePosMatrix[2,2]:=0;
basePosMatrix[3,2]:=0;
basePosMatrix[4,2]:=0;

basePosMatrix[1,3]:=0;
basePosMatrix[2,3]:=0;
basePosMatrix[3,3]:=1;
basePosMatrix[4,3]:=0;

basePosMatrix[1,4]:=x;
basePosMatrix[2,4]:=y;
basePosMatrix[3,4]:=z;
basePosMatrix[4,4]:=1;

//***************output1:C5 posture relative to origin(other than C0)*************//
c14:=COS(q1+q4); s14:=SIN(q1+q4); 
c5:=COS(q5); s5:=SIN(q5);
c1:=COS(q1); s1:=SIN(q1);

T_50[1,1]:=c14*c5; 
T_50[2,1]:=s14*c5; 
T_50[3,1]:=-s5; 
T_50[4,1]:=0;

T_50[1,2]:=-c14*s5;
T_50[2,2]:=-s14*s5; 
T_50[3,2]:=-c5; 
T_50[4,2]:=0;

T_50[1,3]:=-s14;
T_50[2,3]:=c14;
T_50[3,3]:=0;
T_50[4,3]:=0;

T_50[1,4]:=a2*c1 + q2*s1;
T_50[2,4]:=a2*s1 - q2*c1;
T_50[3,4]:=d4 + q3;
T_50[4,4]:=1;

matMultiply(basePosMatrix,T_50,F5);
r_cartPose.m_pos[1]:=F5[1,4]; r_cartPose.m_pos[2]:=F5[2,4]; r_cartPose.m_pos[3]:=F5[3,4];

r_cartPose.m_rot[1,1]:=F5[1,1];  r_cartPose.m_rot[1,2]:=F5[1,2];  r_cartPose.m_rot[1,3]:=F5[1,3];
r_cartPose.m_rot[2,1]:=F5[2,1];  r_cartPose.m_rot[2,2]:=F5[2,2];  r_cartPose.m_rot[2,3]:=F5[2,3];
r_cartPose.m_rot[3,1]:=F5[3,1];  r_cartPose.m_rot[3,2]:=F5[3,2];  r_cartPose.m_rot[3,3]:=F5[3,3];

//********************output2:remote center position************************//
fixPointTransform[1,1]:=1;  fixPointTransform[2,2]:=1;  fixPointTransform[3,3]:=1;  fixPointTransform[4,4]:=1;  
fixPointTransform[2,4]:=-d6;  
matMultiply(F5,fixPointTransform,fixPointMatrix);
r_rcPos[1]:=fixPointMatrix[1,4];  r_rcPos[2]:=fixPointMatrix[2,4];  r_rcPos[3]:=fixPointMatrix[3,4];
END_METHOD

METHOD PUBLIC init : BOOL
VAR_INPUT
	i_armIdx:INT;
END_VAR
VAR 
	i :INT ;
	currentRatioMotor2Jnt:LREAL;
END_VAR
// arm statues init
m_armIdx:=i_armIdx;

// joint init
FOR i:=1 TO g_setupJntNum DO
	m_joints[i].init(m_armIdx, i,g_setupArmCtrlCycleTime);
END_FOR

// joint init
FOR i:=1 TO g_setupJntNum DO
	m_joints[i].initJntPos();
END_FOR

// update arm status if joint position is re-init
updateStatus();

// joint controller init
FOR i:=1 TO g_setupJntNum DO 
	currentRatioMotor2Jnt:=GVL_SetupMotorParameters.g_motorTrqConst[i]*GVL_SetupMotorParameters.g_motorReduction[i]/1000;
	m_jntPIDCtrl[i].init(g_setupArmCtrlCycleTime,GVL_SetupControlParameters.g_posKp[i],GVL_SetupControlParameters.g_posKd[i],
		GVL_SetupControlParameters.g_posKi[i], GVL_SetupControlParameters.g_posKiLimit[i]* currentRatioMotor2Jnt,
		GVL_SetupControlParameters.g_posCtrlLimit[i]*currentRatioMotor2Jnt);
END_FOR

//init arm netID and adrr
m_armNetId := GVL_SlaveJointEncoderCaliData.g_slaveArmNetID[armIdx];
m_jointAddrJ8 := GVL_SlaveJointEncoderCaliData.g_slaveJointNetPort[armIdx,3];
m_jointAddrPbox := GVL_SlaveJointEncoderCaliData.g_slaveJointNetPort[armIdx,4];
END_METHOD

METHOD PUBLIC isEnabled : BOOL
VAR_IN_OUT CONSTANT
	i_jntIdx :Vec5i;
END_VAR
VAR
	i :INT ;
END_VAR
isEnabled := TRUE;
FOR i:=1 TO g_setupJntNum DO
	IF 1= i_jntIdx[i] THEN
		isEnabled :=  (m_joints[i].isEnabled() AND isEnabled);
	END_IF
END_FOR
END_METHOD

PROPERTY jnt5AdjustDir : int
GET
jnt5AdjustDir := m_jnt5AdjustDir;
END_GET
END_PROPERTY

PROPERTY jntGravity :REFERENCE TO Vec5d
GET
jntGravity ref=m_jntGravity;
END_GET
END_PROPERTY

PROPERTY manualAdjustOn : bool
GET
manualAdjustOn := m_manualAdjustOnFlag;
END_GET
END_PROPERTY

PROPERTY rawJntCurrent :REFERENCE TO Vec5d
GET
rawJntCurrent ref=m_rawJntCurrent;
END_GET
END_PROPERTY

PROPERTY rcPos :REFERENCE to Vec3d
GET
rcPos REF= m_rcPos;
END_GET
END_PROPERTY

// update joints control command
METHOD PUBLIC updateCmds : BOOL
VAR_IN_OUT CONSTANT
	i_armCtrlCmd : ST_SetupArmCtrlCmds;
END_VAR
VAR
	i:INT;
END_VAR
m_cmdJntTrq:=i_armCtrlCmd.m_cmdJntTrq;
m_cmdJntPos :=i_armCtrlCmd.m_cmdJntPos;
m_cmdJntVel :=i_armCtrlCmd.m_cmdJntVel;

// enable/disable joints
enable(i_armCtrlCmd.m_jntEnableFlag);

// position/torque control
FOR i:=1 TO g_setupJntNum DO 
	IF i_armCtrlCmd.m_jntOPMode[i]=DriverOPMode_PosTrq THEN
		// position controller and gravity feedforward
		m_cmdJntTrq[i]:=m_jntPIDCtrl[i].run(m_cmdJntPos[i],m_curJntPos[i],0,m_curJntVel[i]);
		m_cmdJntTrq[i]:=m_cmdJntTrq[i]+m_jntGravity[i];
		m_joints[i].updateCmds(DriverOPMode_Trq,m_cmdJntPos[i],m_cmdJntTrq[i]);
	ELSIF i_armCtrlCmd.m_jntOPMode[i]=DriverOPMode_Trq THEN
		// gravity feedforward
		m_jntPIDCtrl[i].reset();
		m_cmdJntTrq[i]:=m_cmdJntTrq[i]+m_jntGravity[i]+GVL_SetupArmDynamics.g_setupJntGravityOffset[m_armIdx, i];
		m_joints[i].updateCmds(DriverOPMode_Trq,i_armCtrlCmd.m_cmdJntPos[i],m_cmdJntTrq[i]);
	ELSE
		m_jntPIDCtrl[i].reset();
		m_cmdJntTrq[i]:=0;
		m_joints[i].updateCmds(DriverOPMode_Pos,i_armCtrlCmd.m_cmdJntPos[i],m_cmdJntTrq[i]);
	END_IF
	
END_FOR
END_METHOD

METHOD PUBLIC updateDyna : BOOL
VAR_IN_out constant
	i_jnt3Gravity :LREAL;
	i_jnt5Gravity :LREAL;
END_VAR
m_jntGravity[3]:=i_jnt3Gravity;
m_jntGravity[5]:=i_jnt5Gravity;
END_METHOD

// update arm status, including kinematic and dynamic
METHOD PUBLIC updateStatus : BOOL
VAR_INPUT
END_VAR
VAR 
	i,j:INT;
END_VAR
// update joint data
FOR i:=1 TO g_setupJntNum DO
	m_joints[i].updateStatus();
END_FOR

// check adjust button
checkIO();

// get joint data
FOR i:=1 TO g_setupJntNum DO
	m_curMotorPos[i]:=m_joints[i].motorPos;
	m_curLinkPos[i]:=m_joints[i].linkPos;
	m_curJntPos[i]:=m_joints[i].jntPos;
	m_curJntVel[i]:=m_joints[i].jntVel;
	m_curJntTrq[i]:=m_joints[i].jntTrq;
	m_rawJntCurrent[i]:=m_joints[i].rawCurrent;
	m_filtJntCurrent[i]:=m_joints[i].filtCurrent;
	m_cmdJntCurrent[i]:=m_joints[i].cmdCurrent;
END_FOR 

// cartesion pose
forwardKinematic(m_curJntPos,m_curCartPose,m_rcPos);
END_METHOD

END_FUNCTION_BLOCK

// ---- FBs_Robots/FB_SetupJoint.TcPOU
FUNCTION_BLOCK FB_SetupJoint EXTENDS FB_JointBase
VAR_INPUT
END_VAR
VAR_OUTPUT
END_VAR
VAR
END_VAR

METHOD PUBLIC init : BOOL
VAR_INPUT
	i_armIdx :INT;
	i_jntIdx :INT;
	i_controlCycleTime :LREAL;
END_VAR
m_armIdx:=i_armIdx;
m_jntIdx:=i_jntIdx;
m_cycleTime := i_controlCycleTime;

// hardware parameters
m_motorEncoderRes :=GVL_SetupMotorParameters.g_incEncoderRes[i_jntIdx];
m_linkEncoderRes :=GVL_SetupMotorParameters.g_absEncoderRes[i_jntIdx];
m_motorReduction :=GVL_SetupMotorParameters.g_motorReduction[i_jntIdx];
m_linkEncoderReduction :=GVL_SetupMotorParameters.g_absEncoderReduction[i_jntIdx];
m_trqConst :=GVL_SetupMotorParameters.g_motorTrqConst[i_jntIdx];
m_maxCurrent :=GVL_SetupMotorParameters.g_motorMaxCurrent[i_jntIdx];
m_motorDir :=GVL_SetupMotorParameters.g_motorDir[i_jntIdx];								
m_minJntPos	:=GVL_SetupMotorParameters.g_minJntPos[m_armIdx,i_jntIdx];
m_maxJntPos	:=GVL_SetupMotorParameters.g_maxJntPos[m_armIdx,i_jntIdx];

//link encoder calibartion data
m_linkEncoderDir :=GVL_SetupJointEncoderCaliData.g_asbEncoderDir[i_jntIdx];
m_minLinkEncoder :=GVL_SetupJointEncoderCaliData.g_minLinkEncoder[i_armIdx, i_jntIdx] - m_linkEncoderDir*GVL_SetupJointEncoderCaliData.g_linkEncLimitBuffer; // expand limit
m_maxLinkEncoder :=GVL_SetupJointEncoderCaliData.g_maxLinkEncoder[i_armIdx, i_jntIdx] + m_linkEncoderDir*GVL_SetupJointEncoderCaliData.g_linkEncLimitBuffer; // expand limit
m_caliLinkEncoder :=GVL_SetupJointEncoderCaliData.g_caliLinkEncoder[i_armIdx, i_jntIdx];
m_linkEncCaliJntPos :=GVL_SetupJointEncoderCaliData.g_linkEncCaliJntPos[i_armIdx,i_jntIdx];
m_linkEncZeroCross :=GVL_SetupJointEncoderCaliData.g_linkEncZeroCross[i_armIdx, i_jntIdx];
m_multiCycles :=GVL_SetupJointEncoderCaliData.g_multipleCyclesJoint[i_armIdx,i_jntIdx];

// convert cali link encoder if joint cross zero
IF 1=m_linkEncZeroCross THEN
	IF 1=m_linkEncoderDir AND m_caliLinkEncoder < m_minLinkEncoder THEN
		m_caliLinkEncoder := GVL_SetupJointEncoderCaliData.g_caliLinkEncoder[i_armIdx, i_jntIdx] + m_linkEncoderRes;
	ELSIF -1=m_linkEncoderDir AND m_caliLinkEncoder < m_maxLinkEncoder THEN
		m_caliLinkEncoder := GVL_SetupJointEncoderCaliData.g_caliLinkEncoder[i_armIdx, i_jntIdx] + m_linkEncoderRes;
	END_IF
END_IF

// macro data
m_trq2CurrentRatio:=m_motorDir * 1000.0/(m_trqConst*m_motorReduction);
m_current2TrqRatio:=m_motorDir * (m_trqConst*m_motorReduction)/1000.0;
m_linkEnc2PosRatio := 2*PI*m_linkEncoderDir/(m_linkEncoderReduction*m_linkEncoderRes);
m_motorEnc2PosRatio := 2*PI * m_motorDir/(m_motorReduction * m_motorEncoderRes);

// motor data init
m_rawJntVel :=0;
m_curJntVel:=0;
m_curJntTrq :=0;
m_rawCurrent :=0;
m_filtCurrent :=0;
m_cmdJntVel :=0.0;
m_cmdJntTrq :=0.0;
m_cmdCurrent := 0.0;

// filter init
m_jntVelLpf.init(1, GVL_SetupControlParameters.g_curJntVelLpfCutoffFreq, g_setupArmCtrlFreq);
m_cmdTrqLpf.init(1, GVL_SetupControlParameters.g_cmdJntTrqLpfCutoffFreq, g_setupArmCtrlFreq);
m_curTrqLpf.init(1, GVL_SetupControlParameters.g_curJntTrqLpfCutoffFreq, g_setupArmCtrlFreq);

// driver init value
m_motorOutputs.m_controlWord:=DriverCtrlWord_INIT;
m_motorOutputs.m_opMode:=INT_TO_SINT(DriverOPMode_Pos);
m_motorOutputs.m_cmdCurrent:=0;
m_motorOutputs.m_cmdMotorEncoder:=m_motorInputs.m_motorEncoder;
END_METHOD

METHOD PUBLIC updateStatus : BOOL
VAR_INPUT
END_VAR
// compute joint position
m_curLinkPos:= linkEnc2Pos();
m_curMotorPos:=motorEnc2Pos();
m_curLinkSingle := m_curLinkPos - 2*PI* m_linkEncCycles;

// setup joint1/2 have no motor, use link position
// joint3 use link position to get a more sensitive reaction during adjust
IF m_jntIdx <= 3 THEN
	m_curJntPos := m_curLinkPos;
ELSE
	m_curJntPos := m_curMotorPos;
END_IF

// compute joint velocity
m_curVelCalCycles := m_curVelCalCycles+1;
IF m_curVelCalCycles > m_velCalcCycles THEN
	m_rawJntVel:= (m_curJntPos-m_lastJntPos)/(m_cycleTime*m_velCalcCycles);
	m_curJntVel := m_jntVelLpf.run(m_rawJntVel);
	m_lastJntPos :=m_curJntPos;	
	m_curVelCalCycles:=1;
END_IF


// current and torque
m_rawCurrent := m_motorInputs.m_current;
m_filtCurrent := m_curTrqLpf.run(m_rawCurrent);
m_curJntTrq := m_filtCurrent * m_current2TrqRatio;
END_METHOD

END_FUNCTION_BLOCK

// ---- FBs_Robots/FB_SetupRobot.TcPOU
FUNCTION_BLOCK FB_SetupRobot
VAR_INPUT
END_VAR
VAR_OUTPUT
END_VAR
VAR
	// setup arms, responsible for arm kinematic and control
	m_setupArms :ARRAY[1..g_sArmNum] OF FB_SetupArm;
	
	// arm light control word
	m_lightCrlWord :ARRAY [1..g_sArmNum] OF UDINT;
	
	// arm state
	m_setupArmState:ARRAY[1..g_sArmNum] OF E_setupArmState:=[4(E_setupArmState.SetupArmState_Error)];
	m_lastSetupArmState:ARRAY[1..g_sArmNum] OF E_setupArmState:=[4(E_setupArmState.SetupArmState_Error)];
	m_nextSetupArmState:ARRAY[1..g_sArmNum] OF E_setupArmState:=[4(E_setupArmState.SetupArmState_Error)];
	
	// all arm controller instance 
	m_armCtrlFactory :ARRAY[1..g_sArmNum,1..SetupArmState_totalNum] OF I_SetupArmCtrl;
	m_armInit :ARRAY[1..g_sArmNum] OF FB_SetupCtrlInit;
	m_armError :ARRAY[1..g_sArmNum] OF FB_SetupCtrlError;
	m_armSelfCheck :ARRAY[1..g_sArmNum] OF FB_SetupCtrlSelfCheck;
	m_armHold :ARRAY[1..g_sArmNum] OF FB_SetupCtrlHold;
	m_armManualAdjust :ARRAY[1..g_sArmNum] OF FB_SetupCtrlManualAdjust;
	m_armAutoAdjust :ARRAY[1..g_sArmNum] OF FB_SetupCtrlAutoAdjust;
	m_armPackage :ARRAY[1..g_sArmNum] OF FB_SetupCtrlPackage;
	m_armCart :ARRAY[1..g_sArmNum] OF FB_SetupCtrlCart;
	m_armJnt3GraCali :ARRAY[1..g_sArmNum] OF FB_SetupCtrlJnt3GraCali;
	m_armJnt5GraCali :ARRAY[1..g_sArmNum] OF FB_SetupCtrlJnt5GraCali;
	m_armDisable :ARRAY[1..g_sArmNum] OF FB_SetupCtrlDisable;
	m_Performance :ARRAY[1..g_sArmNum] OF FB_SetupCtrlPerformance;
	
	
	// arm controller interface
	m_armCtrl :ARRAY[1..g_sArmNum] OF I_SetupArmCtrl;
	m_armCtrlCmds :ARRAY[1..g_sArmNum] OF ST_SetupArmCtrlCmds;

END_VAR

METHOD PROTECTED controllerTransit : BOOL
VAR_INPUT
END_VAR
VAR
	i:int;
END_VAR
FOR i:=1 TO g_sArmNum DO 
	// Controller transit
	IF m_nextSetupArmState[i]<> m_setupArmState[i] THEN
		// reset current controller
		m_armCtrl[i].reset();
		
		// transit to new controller
		m_lastSetupArmState[i]:=m_setupArmState[i];
		m_setupArmState[i]:=m_nextSetupArmState[i];
		m_armCtrl[i]:=m_armCtrlFactory[i,m_setupArmState[i]];
		
		// init next controller
		m_armCtrl[i].Init(m_setupArms[i],m_armCtrlCmds[i]);
		m_setupArms[i].updateCmds(m_armCtrlCmds[i]);
	END_IF
END_FOR
END_METHOD

METHOD PUBLIC getStatus : BOOL
VAR_IN_OUT
	// slave robot information, including arm status and cartesian data
	r_setupStatus :ST_SetupStatus;
	
	// slave robot joint data
	r_setupJointsData :ST_SetupJointData;
	
END_VAR

VAR
	i:INT;
END_VAR
r_setupStatus.m_armState:=m_setupArmState;

// TODO: project cartesion data to monitor coordinate
FOR i:=1 TO g_sArmNum DO
	
	// cartesion
	r_setupStatus.m_curEndPose[i]:=m_setupArms[i].curCartPose;
	r_setupStatus.m_rcPos[i]:=m_setupArms[i].rcPos;
	
	// joint
	r_setupJointsData.m_curMotorPos[i]:=m_setupArms[i].curMotorPos;
	r_setupJointsData.m_curLinkPos[i]:=m_setupArms[i].curLinkPos;
	r_setupJointsData.m_curJntPos[i]:=m_setupArms[i].curJntPos;
	r_setupJointsData.m_curJntVel[i]:=m_setupArms[i].curJntVel;
	r_setupJointsData.m_rawJntCurrent[i]:=m_setupArms[i].rawJntCurrent;
	r_setupJointsData.m_cmdJntCurrent[i]:=m_setupArms[i].cmdJntCurrent;
	r_setupJointsData.m_cmdJntVel[i]:=m_setupArms[i].m_cmdJntVel;
	
	// command info
	// joint info
	r_setupJointsData.m_cmdJntPos[i]:=m_armCtrlCmds[i].m_cmdJntPos;
	
END_FOR
END_METHOD

METHOD PUBLIC Init : BOOL
VAR_INPUT
END_VAR
VAR
	i:INT;
END_VAR
FOR i:=1 TO g_sArmNum DO
	// arm init
	m_setupArms[i].Init(i);
	m_setupArmState[i]:=SlaveArmState_Init;
	m_lastSetupArmState[i]:=SlaveArmState_Init;
	m_nextSetupArmState[i]:=SlaveArmState_Init;
	
	// command init
	m_armCtrlCmds[i].m_jntEnableFlag := g_zeroVec5i;
	m_armCtrlCmds[i].m_jntOPMode := g_setupAllPosMode;
	m_armCtrlCmds[i].m_cmdJntPos := m_setupArms[i].curJntPos;
	m_armCtrlCmds[i].m_cmdJntVel := g_zeroVec5d;
	m_armCtrlCmds[i].m_cmdJntAcc := g_zeroVec5d;
	m_armCtrlCmds[i].m_cmdJntTrq := g_zeroVec5d;
	
	// generate controller factory
	m_armCtrlFactory[i,SetupArmState_Error] := m_armError[i];
	m_armCtrlFactory[i,SetupArmState_Init] := m_armInit[i];
	m_armCtrlFactory[i,SetupArmState_SelfCheck] := m_armSelfCheck[i];
	m_armCtrlFactory[i,SetupArmState_Hold] := m_armHold[i];
	m_armCtrlFactory[i,SetupArmState_ManualAdjust] := m_armManualAdjust[i];
	m_armCtrlFactory[i,SetupArmState_AutoAdjust] := m_armAutoAdjust[i];
	m_armCtrlFactory[i,SetupArmState_Package] := m_armPackage[i];
	m_armCtrlFactory[i,SetupArmState_Cart] := m_armCart[i];
	m_armCtrlFactory[i,SetupArmState_jnt3GravityCali] := m_armJnt3GraCali[i];
	m_armCtrlFactory[i,SetupArmState_jnt5GravityCali] := m_armJnt5GraCali[i];
	m_armCtrlFactory[i,SetupArmState_Disable] := m_armDisable[i];
	m_armCtrlFactory[i,SetupArmState_Performance] := m_Performance[i];
	
	// assign controller
	m_armCtrl[i]:=m_armCtrlFactory[i,m_setupArmState[i]];
	m_armCtrl[i].Init(m_setupArms[i],m_armCtrlCmds[i]);
END_FOR
END_METHOD

METHOD PUBLIC run : BOOL
VAR_IN_OUT CONSTANT
	i_setupInputDataPool:ST_SetupInputDataPool;
END_VAR
VAR
	i:INT;
END_VAR
// update arm status
FOR i:=1 TO g_sArmNum DO
	// update dynamic data
	m_setupArms[i].updateDyna(i_setupInputDataPool.m_setupJnt3Gravity[i], i_setupInputDataPool.m_setupJnt5Gravity[i]);
								
	// update slave arm kinematics
	m_setupArms[i].updateStatus();
END_FOR

// state machine transition
stateMachine(i_setupInputDataPool);

//update arm light
updateArmLight(i_setupInputDataPool);

// controller transition
controllerTransit();

FOR i:=1 TO g_sArmNum DO
	// null ptr check
	ASSERT(0 <> m_armCtrl[i]);
	
	// run controller
	m_armCtrl[i].run(m_setupArms[i],m_armCtrlCmds[i]);

	// update commands to drivers
	m_setupArms[i].updateCmds(m_armCtrlCmds[i]);
END_FOR
END_METHOD

// state machine check and transit 
METHOD PROTECTED stateMachine : BOOL
VAR_IN_OUT CONSTANT
		i_setupInputDataPool:ST_SetupInputDataPool;
END_VAR
VAR
	i:INT;
END_VAR
FOR i:=1 TO g_sArmNum DO
	// State machine transit 
	CASE m_setupArmState[i] OF
		// error
		SetupArmState_Error:
			IF FALSE = i_setupInputDataPool.m_safetyData.m_setupErrFlag[i]  THEN
				m_nextSetupArmState[i]:=SetupArmState_Hold;
			END_IF
			// to manual adjust
			//IF m_setupArms[i].manualAdjustOn OR m_setupArms[i].m_jnt5AdjustDir<>0 THEN
			IF m_setupArms[i].manualAdjustOn THEN
				m_nextSetupArmState[i]:=SetupArmState_ManualAdjust;
			END_IF
			
		// init
		SetupArmState_Init:
			// to hold. No self check for setup arm currently
			IF m_armCtrl[i].isFinished  THEN
				m_nextSetupArmState[i]:=SetupArmState_Hold;
			END_IF

		//self check
		SetupArmState_SelfCheck:
			IF m_armCtrl[i].isFinished  THEN
				m_nextSetupArmState[i]:=SetupArmState_Hold;
			END_IF
		
		//hold
		SetupArmState_Hold:
			// to manual adjust
			IF m_setupArms[i].manualAdjustOn OR m_setupArms[i].m_jnt5AdjustDir<>0 THEN
				m_nextSetupArmState[i]:=SetupArmState_ManualAdjust;
			END_IF
			
		
		// manual adjust
		SetupArmState_ManualAdjust:
			// to hold
			IF NOT(m_setupArms[i].manualAdjustOn) AND m_setupArms[i].jnt5AdjustDir=0 THEN
				m_nextSetupArmState[i] := SetupArmState_Hold;
			END_IF
			
		// auto adjust
		SetupArmState_AutoAdjust:
				
		//package
		SetupArmState_Package:
		
		//cart
		SetupArmState_Cart:
		
		//joint 5 gravity calibration
		SetupArmState_jnt5GravityCali:
			IF m_armCtrl[i].isFinished  THEN
				m_nextSetupArmState[i]:=SetupArmState_Hold;
			END_IF 
			
		//joint 3 gravity calibration
		SetupArmState_jnt3GravityCali:
			IF m_armCtrl[i].isFinished  THEN
				m_nextSetupArmState[i]:=SetupArmState_Hold;
			END_IF 
		
		// arm disable
		SetupArmState_Disable:
			IF NOT(SlaveArmControl.m_slaveInputDataPool.m_UIData.m_slaveArmDisableFlag[i]) THEN
				m_nextSetupArmState[i]:= SetupArmState_Hold;
			END_IF
			
		//arm Performance
		SetupArmState_Performance:
			// to hold
			IF  m_armCtrl[i].isFinished THEN
				m_nextSetupArmState[i]:=SetupArmState_Hold;
			END_IF				
	END_CASE
	
	// arm disable
	IF SlaveArmControl.m_slaveInputDataPool.m_UIData.m_slaveArmDisableFlag[i] THEN
		m_nextSetupArmState[i] := SetupArmState_Disable;
	// error check
	//ELSIF. i_setupInputDataPool.m_safetyData.m_setupErrFlag[i] AND NOT (m_setupArms[i].manualAdjustOn OR m_setupArms[i].m_jnt5AdjustDir<>0) THEN
	ELSIF i_setupInputDataPool.m_safetyData.m_setupErrFlag[i] AND NOT (m_setupArms[i].manualAdjustOn) THEN
		m_nextSetupArmState[i]:=SetupArmState_Error;
	END_IF
END_FOR
END_METHOD

METHOD updateArmLight : BOOL
VAR_IN_OUT CONSTANT
	i_setupInputDataPool:ST_SetupInputDataPool;
END_VAR

VAR
	i : INT;
	slaveArmState :E_SlaveArmState;
END_VAR
//*******************机械臂与动力盒上的灯光写入********************
//不可恢复性故障-----红色常亮
//可恢复故障----琥珀色-先闪烁5s、再进行常亮
//正处于器械控制或者端口控制状态-----蓝色闪烁
//该手术臂正在执行一项需要用户短时间等待的活动、例如器械卡接----蓝色-脉动闪烁
//工具更换引导正在进行中-----绿色闪烁
//未通电、已禁用、已收起----------关
//系统正常运行-----蓝色常亮
//灯光颜色--0-灯灭、1蓝灯常亮、2蓝灯闪烁、3琥珀色闪烁、4红灯闪烁、5绿灯常亮、6绿灯闪烁、7红灯常亮、8琥珀色常亮、9蓝灯脉动式闪烁
FOR i := 1 TO g_sArmNum BY 1 DO
	slaveArmState := i_setupInputDataPool.m_slaveStatus.m_armState[i];
	IF slaveArmState = SlaveArmState_Error OR m_setupArmState[i] = SlaveArmState_Error THEN
		IF SafetyCheck.m_SafetyCheck.m_armErrFlag[i,3] THEN
			m_lightCrlWord[i] := ArmLight_RedBlink;
		ELSIF SafetyCheck.m_SafetyCheck.m_armErrFlag[i,2] THEN
			m_lightCrlWord[i] := ArmLight_AmberBlink;
		END_IF
	ELSIF slaveArmState = SlaveArmState_MountPanel OR slaveArmState = SlaveArmState_MountInstru THEN
		m_lightCrlWord[i] := ArmLight_BluePulse;
	ELSIF slaveArmState = SlaveArmState_InstruRetract OR slaveArmState = SlaveArmState_Adjust OR m_setupArmState[i] = SetupArmState_ManualAdjust THEN
		m_lightCrlWord[i] := ArmLight_BlueBlink;
	ELSIF slaveArmState = SlaveArmState_InstruInvasion THEN
		m_lightCrlWord[i] := ArmLight_GreenBlink;
	ELSIF slaveArmState = SlaveArmState_Disable THEN
		m_lightCrlWord[i] := ArmLight_Off;
	ELSE
		m_lightCrlWord[i] := ArmLight_BlueOn;
	END_IF

	m_setupArms[i].checkLight(m_lightCrlWord[i]);
END_FOR
END_METHOD

END_FUNCTION_BLOCK

// ---- FBs_SetupControllers/FB_SetupCtrlInit.TcPOU
// Brief: Setup Arm Init
FUNCTION_BLOCK PUBLIC FB_SetupCtrlInit EXTENDS FB_SetupArmCtrlBase
VAR_INPUT
END_VAR
VAR_OUTPUT
END_VAR
VAR
	m_initState :INT :=0;
END_VAR

// override this function in each exact controller
METHOD PROTECTED calcCmdJntPos : BOOL
VAR_IN_OUT CONSTANT
	i_setupArm	:FB_SetupArm;
END_VAR


VAR 
	i :INT;
	curJntVel :Vec5d;
END_VAR
IF m_timePeriod > 1.0 then
	m_isFinished :=TRUE;
END_IF
END_METHOD

METHOD PUBLIC init : BOOL
VAR_IN_OUT CONSTANT
	i_setupArm	:FB_SetupArm;
END_VAR
VAR_IN_OUT 
	r_setupArmCtrlCmd :ST_SetupArmCtrlCmds;
END_VAR


VAR
	i:INT;
END_VAR
SUPER^.Init(i_setupArm,r_setupArmCtrlCmd);
END_METHOD

END_FUNCTION_BLOCK

// ---- FBs_SetupControllers/FB_SetupArmCtrlBase.TcPOU
// Setup Arm Base Controller, Hold at Current Posture
FUNCTION_BLOCK FB_SetupArmCtrlBase IMPLEMENTS I_SetupArmCtrl
VAR_INPUT
END_VAR
VAR_OUTPUT
END_VAR
VAR
	// flag if the controller has finished all its jobs
	m_isFinished:BOOL:=FALSE;
	
	// controller execute time period
	m_timePeriod :LREAL:=0;
	
	// arm control data
	m_cmdJntPos : VEC5d;
	m_cmdJntVel : VEC5d;
	m_cmdJntAcc : VEC5d;
	m_cmdJntTrq : VEC5d;
	m_jntOPMode : Vec5i;
	m_jntEnableFlag :Vec5i;
END_VAR

// override this function in each exact controller
METHOD PROTECTED calcCmdJntPos : BOOL
VAR_IN_OUT CONSTANT
	i_setupArm	:FB_SetupArm;
END_VAR
END_METHOD

// override this function in each exact controller
METHOD PROTECTED calcCmdJntTrq : BOOL
VAR_IN_OUT CONSTANT
	i_setupArm	:FB_SetupArm;
END_VAR
// set joint torque to zero in default
m_cmdJntTrq := g_zeroVec5d;
END_METHOD

// override this function in each exact controller
// NOTICE: set joint control mode here, and do some initialization if needed
METHOD PUBLIC init : BOOL
VAR_IN_OUT CONSTANT
	i_setupArm	:FB_SetupArm;
END_VAR
VAR_IN_OUT 
	r_setupArmCtrlCmd :ST_SetupArmCtrlCmds;
END_VAR
m_timePeriod:=0;
m_jntEnableFlag :=g_zeroVec5i;// setup arm joint is diabled by default
m_jntOPMode:=g_setupAllPosMode;
m_cmdJntPos:=i_setupArm.curJntPos;
m_cmdJntVel:=g_zeroVec5d;
m_cmdJntAcc:=g_zeroVec5d;
m_cmdJntTrq:=g_zeroVec5d;

// update commands to arm
r_setupArmCtrlCmd.m_jntEnableFlag :=m_jntEnableFlag;
r_setupArmCtrlCmd.m_cmdJntPos:=m_cmdJntPos;
r_setupArmCtrlCmd.m_cmdJntVel:=m_cmdJntVel;
r_setupArmCtrlCmd.m_cmdJntAcc:=m_cmdJntAcc;
r_setupArmCtrlCmd.m_cmdJntTrq:=m_cmdJntTrq;
r_setupArmCtrlCmd.m_jntOPMode:=m_jntOPMode;
END_METHOD

PROPERTY isFinished : BOOL
GET
isFinished:=m_isFinished;
END_GET
END_PROPERTY

{warning '添加方法实现'}
METHOD reset : BOOL
m_isFinished:=FALSE;
m_timePeriod:=0;
END_METHOD

{warning '添加方法实现'}
METHOD run : BOOL
VAR_IN_OUT CONSTANT
	i_setupArm	:FB_SetupArm;
END_VAR
VAR_IN_OUT 
	r_setupArmCtrlCmd :ST_SetupArmCtrlCmds;
END_VAR

VAR
	i:INT;
END_VAR
IF m_isFinished THEN
	RETURN;
END_IF

// check if arm enabled
IF FALSE = i_setupArm.isEnabled(m_jntEnableFlag) THEN
//	RETURN;
END_IF

// calculate command joint position--Motion control
calcCmdJntPos(i_setupArm);

// calculate command joint torque -- Force control
calcCmdJntTrq(i_setupArm);

// update commands to arm
r_setupArmCtrlCmd.m_jntEnableFlag :=m_jntEnableFlag;
r_setupArmCtrlCmd.m_cmdJntPos:=m_cmdJntPos;
r_setupArmCtrlCmd.m_cmdJntVel:=m_cmdJntVel;
r_setupArmCtrlCmd.m_cmdJntAcc:=m_cmdJntAcc;
r_setupArmCtrlCmd.m_cmdJntTrq:=m_cmdJntTrq;
r_setupArmCtrlCmd.m_jntOPMode:=m_jntOPMode;

// update time period
m_timePeriod := m_timePeriod+g_setupArmCtrlCycleTime;
END_METHOD

END_FUNCTION_BLOCK

// ---- FBs_SetupControllers/FB_SetupCtrlError.TcPOU
// Brief: Setup Arm Error Hold
FUNCTION_BLOCK PUBLIC FB_SetupCtrlError EXTENDS FB_SetupArmCtrlBase
VAR_INPUT
END_VAR
VAR_OUTPUT
END_VAR
VAR
END_VAR

END_FUNCTION_BLOCK

// ---- FBs_SetupControllers/FB_SetupCtrlSelfCheck.TcPOU
// Brief: Setup Arm Self-check
FUNCTION_BLOCK PUBLIC FB_SetupCtrlSelfCheck EXTENDS FB_SetupArmCtrlBase
VAR CONSTANT
	m_selfCheckMotionNum :INT :=1;
END_VAR
VAR
	// slave self-check motion parameters
	m_selfCheckPosture:ARRAY [1..m_selfCheckMotionNum, 1..g_setupJntNum] OF LREAL:=[0.0, 0.0, 0.1, pi/2, PI/2];																			//PI/4, -PI/4, 0.3, pi, pi, pi, pi, pi];
	m_selfCheckMaxjntVel:Vec5d:=[0.1, 0.1, 0.05, 0.1, 0.1];
	m_selfCheckMaxjntAcc:Vec5d:=[0.1, 0.1, 0.25, 0.5, 0.5];
	m_selfCheckMaxjntJerk:Vec5d:=[0.1,0.1, 0.5, 1.0, 1.0];
	
	m_selfCheckTrajIdx: INT := 1;
	m_slefCheckPlanner: ARRAY[1..m_selfCheckMotionNum] OF FB_setupTrajMoveJ;
	
	// collision and safety check threshold
	m_jntCtrlErr:Vec5d;
	m_jntCtrlErrThres :Vec5d:=[2.0*g_deg2rad, 0.005,  0.005, 2(2.0*g_deg2rad)];
	
END_VAR

// override this function in each exact controller
METHOD PROTECTED calcCmdJntPos : BOOL
VAR_IN_OUT CONSTANT
	i_setupArm	:FB_SetupArm;
END_VAR


VAR 
	i :INT;
END_VAR
// check if planner is ready
IF m_slefCheckPlanner[m_selfCheckTrajIdx].isGene = FALSE THEN
	calcCmdJntPos:=FALSE;
	RETURN;
END_IF

// traj plan
calcCmdJntPos :=m_slefCheckPlanner[m_selfCheckTrajIdx].evaluate(m_timePeriod, jntPos=> m_cmdJntPos, jntVel=>m_cmdJntVel, jntAcc=> m_cmdJntAcc);

// check if to transit to next segment
IF(m_timePeriod > m_slefCheckPlanner[m_selfCheckTrajIdx].duration  AND norm(i_setupArm.m_curJntVel)<7*GVL_SlaveControlParameters.g_jntStaticVelThres) THEN
	m_selfCheckTrajIdx:=m_selfCheckTrajIdx+1;
	m_timePeriod:=0;
END_IF

// safety check
vecSub(m_cmdJntPos, i_setupArm.m_curJntPos, m_jntCtrlErr);
FOR i:=1 TO g_setupJntNum DO 
	IF ABS(m_jntCtrlErr[i])> m_jntCtrlErrThres[i] THEN
		m_isFinished:=TRUE;
		RETURN;
	END_IF
END_FOR


// check if to terminated
IF(m_selfCheckTrajIdx > m_selfCheckMotionNum) THEN
	m_isFinished:=TRUE;
END_IF
END_METHOD

METHOD PUBLIC init : BOOL
VAR_IN_OUT CONSTANT
	i_setupArm	:FB_SetupArm;
END_VAR
VAR_IN_OUT 
	r_setupArmCtrlCmd :ST_SetupArmCtrlCmds;
END_VAR


VAR
	i,j :INT;
	startJntPos,endJntPos :Vec5d;
END_VAR
SUPER^.Init(i_setupArm,r_setupArmCtrlCmd);
m_jntEnableFlag[3]:=1;
m_jntEnableFlag[4]:=1;
m_jntEnableFlag[5]:=1;

// traj plan
m_selfCheckTrajIdx :=1;
// fisrt segment
startJntPos:=i_setupArm.curJntPos;
endJntPos := startJntPos;
FOR j:=3 TO 5 DO 
	endJntPos[j]:=m_selfCheckPosture[1,j];
END_FOR
m_slefCheckPlanner[1].init(startJntPos,endJntPos,m_selfCheckMaxjntVel, m_selfCheckMaxjntAcc,m_selfCheckMaxjntJerk);

// other segments
IF m_selfCheckMotionNum>= 2 THEN
	FOR i:=2 TO m_selfCheckMotionNum DO 
		FOR j:=3 TO 5 DO 
			startJntPos[j]:=m_selfCheckPosture[i-1,j];
			endJntPos[j]:=m_selfCheckPosture[i,j];
		END_FOR
		m_slefCheckPlanner[i].init(startJntPos,endJntPos,m_selfCheckMaxjntVel, m_selfCheckMaxjntAcc,m_selfCheckMaxjntJerk);
	END_FOR
END_IF;
END_METHOD

END_FUNCTION_BLOCK

// ---- FBs_TrajectoryPlanning/FB_setupTrajMoveJ.TcPOU
FUNCTION_BLOCK FB_setupTrajMoveJ EXTENDS FB_TrajBase
VAR_OUTPUT
END_VAR
VAR
	// move vector in joint space
	m_startPos:Vec5d;
	m_targetPos:Vec5d;
	m_moveDir : Vec5d;
	m_moveDistance :LREAL;
	
	// doubleS planning for move distance
	m_doubleS :FB_BasicDoubleS;
END_VAR

METHOD evaluate : BOOL
VAR_INPUT
	t :LREAL;
END_VAR

VAR_OUTPUT
	jntPos,jntVel, jntAcc :vec5d;
END_VAR
VAR
	q,q_dot,q_ddot :LREAL;
	moveRange :Vec5d;
END_VAR
evaluate:=m_doubleS.evaluate(t,q=>q,q_dot=>q_dot, q_ddot=>q_dot);
IF evaluate =FALSE THEN
	RETURN;
END_IF

vecMultiNum(m_moveDir,q, moveRange);
vecAdd(moveRange, m_startPos,jntPos);
vecMultiNum(m_moveDir,q_dot, jntVel);
vecMultiNum( m_moveDir,q_ddot, jntAcc);
END_METHOD

METHOD init : BOOL
VAR_INPUT
	i_startJntPos :Vec5d;
	i_targetJntPos :Vec5d;
	i_maxJntVel : Vec5d;
	i_maxJntAcc : Vec5d;
	i_maxJntJerk :Vec5d;
END_VAR
VAR 
	i:INT;
	maxV, maxA, maxJ :LREAL;
	q:ARRAY[1..2] OF LREAL;
	v:ARRAY[1..2] OF LREAL;
END_VAR
m_startPos:=i_startJntPos;
m_targetPos:=i_targetJntPos;
vecSub(i_targetJntPos, i_startJntPos, m_moveDir);
m_moveDistance := norm(m_moveDir);

IF(m_moveDistance<g_smallNum) THEN
	vecMultiNum(g_onesVec7d,1/5, m_moveDir);;
ELSE
	vecMultiNum( m_moveDir,1/m_moveDistance, m_moveDir);
END_IF

// determian max vel/acc/jerk
maxV:=g_largeNum;
maxA:=g_largeNum;
maxJ:=g_largeNum;
FOR i :=1 TO 5 DO 
	IF ABS(m_moveDir[i])>g_smallNum THEN
		maxV := MIN (maxV, ABS(i_maxJntVel[i]/m_moveDir[i]));
		maxA := MIN (maxA, ABS(i_maxJntAcc[i]/m_moveDir[i]));
		maxJ := MIN (maxJ, ABS(i_maxJntJerk[i]/m_moveDir[i]));
	END_IF
END_FOR

// planning for moving distance
q[1]:=0;
q[2]:=m_moveDistance;
v[1]:=0;
v[2]:=0;
m_doubleS.init(q,v, maxV, maxA, maxJ);
m_duration:=m_doubleS.duration;
m_isGenerated:=m_doubleS.isGene;
END_METHOD

END_FUNCTION_BLOCK

// ---- FBs_SetupControllers/FB_SetupCtrlHold.TcPOU
// Brief: Setup Arm Init
FUNCTION_BLOCK PUBLIC FB_SetupCtrlHold EXTENDS FB_SetupArmCtrlBase
VAR_INPUT
END_VAR
VAR_OUTPUT
END_VAR
VAR
	m_initState :INT :=0;
END_VAR

// override this function in each exact controller
METHOD PROTECTED calcCmdJntPos : BOOL
VAR_IN_OUT CONSTANT
	i_setupArm	:FB_SetupArm;
END_VAR


VAR 
	i :INT;
	curJntVel :Vec5d;
END_VAR
// set command joint position to current joint position, it's ok as all the joints is disabled.
// And by doing so, can avoid some fault triggers, like joint control error if joint enter disable too fast and brake can not stop joint immediately. 
IF m_timePeriod < 1.0 THEN
	m_cmdJntPos:=i_setupArm.curJntPos;
END_IF
END_METHOD

// override this function in each exact controller
// NOTICE: set joint control mode here, and do some initialization if needed
METHOD PUBLIC init : BOOL
VAR_IN_OUT CONSTANT
	i_setupArm	:FB_SetupArm;
END_VAR
VAR_IN_OUT 
	r_setupArmCtrlCmd :ST_SetupArmCtrlCmds;
END_VAR
SUPER^.Init(i_setupArm,r_setupArmCtrlCmd);

// TODO: setup joint3 would "jump" a bit when transit from torque mode to position mode
m_jntOPMode[3] := DriverOPMode_Trq;
END_METHOD

END_FUNCTION_BLOCK

// ---- FBs_SetupControllers/FB_SetupCtrlManualAdjust.TcPOU
// Brief: Setup Arm Adjust
FUNCTION_BLOCK PUBLIC FB_SetupCtrlManualAdjust EXTENDS FB_SetupArmCtrlBase
VAR_INPUT
END_VAR
VAR_OUTPUT
END_VAR
VAR
	// friction compensation scale
	m_frictionScale :LREAL :=0.5;
	
	// velocity threshold for friction compensation 
	m_jnt3FrictionCompVelLow :LREAL := 0.0005;
	m_frictionScaleLow :LREAL :=0.3;
	m_jnt3FrictionCompVelMiddle :LREAL := 0.005;
	m_frictionScaleMiddle :LREAL :=0.5;
	m_jnt3FrictionCompVelHigh :LREAL := 0.05;
	m_frictionScaleHigh :LREAL :=0.7;
	
	// jnt5 adjust velocity
	m_jnt5MaxAdjustVel :LREAL:=5.0*g_deg2Rad;
	m_jnt5MaxAdjustAcc :LREAL:=60*g_deg2Rad;
	
	// jnt5 enabled time period
	m_jnt5EnableTime :LREAL :=0;
	
	// time threshold to drive jnt5 after it's enabled
	m_jnt5AdjustWaitTime :LREAL := 0.25;

	// distance buffer from joint limit to start damp
	m_limitBufferForDamp :LREAL :=0.05;
	
	// max damp
	m_maxDamp :LREAL := 3000;
	
	m_limitBufferForCtrl : LREAL := 0.01;
END_VAR

// override this function in each exact controller
METHOD PROTECTED calcCmdJntPos : BOOL
VAR_IN_OUT CONSTANT
	i_setupArm	:FB_SetupArm;
END_VAR


VAR 
	i :INT;
END_VAR
// enable/disenable joint5
IF i_setupArm.jnt5AdjustDir = 0 THEN
	m_jntEnableFlag[5] := 0;
	m_cmdJntPos[5]:=i_setupArm.curJntPos[5];
	m_jnt5EnableTime:=0;
	m_cmdJntVel[5]:=0;
	RETURN;
ELSE
	// disable joints if this joint is an unrecoverable failure
	m_jntEnableFlag[5] :=  BOOL_TO_INT( NOT (SafetyCheck.m_SafetyCheck.m_jntErrFlag[i_setupArm.armIdx, 0, 3] OR  SafetyCheck.m_SafetyCheck.m_jntErrFlag[i_setupArm.armIdx, 5, 3]));
	m_jnt5EnableTime := m_jnt5EnableTime + g_setupArmCtrlCycleTime;
END_IF

// update command position
IF m_jnt5EnableTime>m_jnt5AdjustWaitTime THEN
	m_cmdJntVel[5]:=m_cmdJntVel[5] + i_setupArm.jnt5AdjustDir * m_jnt5MaxAdjustAcc * g_setupArmCtrlCycleTime;
	m_cmdJntVel[5]:=LIMIT(-m_jnt5MaxAdjustVel, m_cmdJntVel[5], m_jnt5MaxAdjustVel);
	
	// joint limit
	IF (m_cmdJntPos[5] > GVL_SetupMotorParameters.g_maxJntPos[i_setupArm.armIdx, 5] - g_setupJntPosLimitBuffer[5] AND m_cmdJntVel[5]>0) OR 
		(m_cmdJntPos[5] < GVL_SetupMotorParameters.g_minJntPos[i_setupArm.armIdx, 5] + g_setupJntPosLimitBuffer[5] AND m_cmdJntVel[5]<0)  THEN
		m_cmdJntVel[5] := 0;
	END_IF
	
	m_cmdJntPos[5]:= m_cmdJntPos[5] + m_cmdJntVel[5] * g_setupArmCtrlCycleTime;
END_IF
END_METHOD

// override this function in each exact controller
METHOD PROTECTED calcCmdJntTrq : BOOL
VAR_IN_OUT CONSTANT
	i_setupArm	:FB_SetupArm;
END_VAR
VAR
	i:INT;
	vel :LREAL;
	scale:LREAL;
	ratio:LREAL;
	dampScale :LREAL;
	limitDis:LREAL;
	dampOffset : LREAL;
END_VAR
// set joint torque to zero in default
m_cmdJntTrq := g_zeroVec5d;

//enable/diable  joint1-4
IF NOT(i_setupArm.manualAdjustOn) THEN
	FOR i:=1 TO 4 DO
		m_jntEnableFlag[i] := 0;
		m_jntOPMode[i]:=DriverOPMode_Pos;
	END_FOR
	
	// TODO: setup joint3 would "jump" a bit when transit from torque mode to position mode
	m_jntOPMode[3] := DriverOPMode_Trq;
	RETURN;
ELSE
	FOR i:=1 TO 4 DO
		// disable joints if this joint is an unrecoverable failure
		m_jntEnableFlag[i] := BOOL_TO_INT( NOT (SafetyCheck.m_SafetyCheck.m_jntErrFlag[i_setupArm.armIdx, 0, 3] OR  SafetyCheck.m_SafetyCheck.m_jntErrFlag[i_setupArm.armIdx, i, 3]));
		m_jntOPMode[i]:=DriverOPMode_Trq;
		m_cmdJntPos[i] := i_setupArm.curJntPos[i];
	END_FOR
END_IF

// friction scale
vel:=ABS(i_setupArm.curJntVel[3]);
IF vel < m_jnt3FrictionCompVelLow THEN
	m_frictionScale := m_frictionScaleLow * vel/m_jnt3FrictionCompVelLow ;
ELSIF  vel > m_jnt3FrictionCompVelLow AND vel  < m_jnt3FrictionCompVelMiddle THEN
	ratio:= (vel-m_jnt3FrictionCompVelLow)/(m_jnt3FrictionCompVelMiddle-m_jnt3FrictionCompVelLow);
	m_frictionScale :=m_frictionScaleLow+ratio * (m_frictionScaleMiddle-m_frictionScaleLow);
ELSIF  vel > m_jnt3FrictionCompVelMiddle AND vel  < m_jnt3FrictionCompVelHigh THEN
	ratio:= (vel-m_jnt3FrictionCompVelMiddle)/(m_jnt3FrictionCompVelHigh-m_jnt3FrictionCompVelMiddle);
	m_frictionScale :=m_frictionScaleMiddle+ratio * (m_frictionScaleHigh-m_frictionScaleMiddle);
ELSIF  vel > m_jnt3FrictionCompVelHigh THEN
	m_frictionScale := m_frictionScaleHigh;
END_IF

// add damp near joint limit 
IF (i_setupArm.curJntPos[3] > GVL_SetupMotorParameters.g_maxJntPos[1,3] - m_limitBufferForCtrl ) 
	OR (i_setupArm.curJntPos[3] < GVL_SetupMotorParameters.g_minJntPos[1,3] + m_limitBufferForCtrl) OR CartControl.m_cartRobot.m_slaveCart.m_columnAdjustEnable  THEN
	dampOffset:= 0;
ELSIF (i_setupArm.curJntPos[3] > GVL_SetupMotorParameters.g_maxJntPos[1,3] - m_limitBufferForDamp AND  i_setupArm.curJntVel[3]> 0 ) 
	OR (i_setupArm.curJntPos[3] < GVL_SetupMotorParameters.g_minJntPos[1,3] + m_limitBufferForDamp AND  i_setupArm.curJntVel[3]<0 )  THEN
	limitDis := MIN(GVL_SetupMotorParameters.g_maxJntPos[1,3] - i_setupArm.curJntPos[3], i_setupArm.curJntPos[3]-GVL_SetupMotorParameters.g_minJntPos[1,3]);
	dampScale  :=LIMIT(0, 1-limitDis/(m_limitBufferForDamp-m_limitBufferForCtrl),1);
	dampOffset:= -dampScale * m_maxDamp * i_setupArm.curJntVel[3];
END_IF


// add friction compensation
m_frictionScale := LIMIT(0, m_frictionScale, 1);
m_cmdJntTrq[3]:= m_frictionScale * sign(i_setupArm.curJntVel[3])*jnt3Friction(i_setupArm.armIdx, i_setupArm.curJntPos[3]) + dampOffset;
END_METHOD

METHOD PUBLIC init : BOOL
VAR_IN_OUT CONSTANT
	i_setupArm	:FB_SetupArm;
END_VAR
VAR_IN_OUT 
	r_setupArmCtrlCmd :ST_SetupArmCtrlCmds;
END_VAR
SUPER^.Init(i_setupArm,r_setupArmCtrlCmd);
m_jnt5EnableTime :=0;
END_METHOD

METHOD PROTECTED jnt3Friction : Lreal
VAR_INPUT
	i_armIdx:INT;
	i_jnt3Pos :LREAL;
END_VAR

VAR
	q:LREAL;
END_VAR
q := LIMIT(GVL_SetupArmDynamics.g_setupJnt3GravityPosRange[i_armIdx,1], i_jnt3Pos, GVL_SetupArmDynamics.g_setupJnt3GravityPosRange[i_armIdx,2]);
jnt3Friction:=GVL_SetupArmDynamics.g_setupJnt3FrictionParams[i_armIdx,1]*EXPT(q,3)+GVL_SetupArmDynamics.g_setupJnt3FrictionParams[i_armIdx,2]*EXPT(q,2)+
				GVL_SetupArmDynamics.g_setupJnt3FrictionParams[i_armIdx,3]*q+GVL_SetupArmDynamics.g_setupJnt3FrictionParams[i_armIdx,4];
END_METHOD

END_FUNCTION_BLOCK

// ---- FBs_SetupControllers/FB_SetupCtrlAutoAdjust.TcPOU
// Brief: Setup Arm Adjust
FUNCTION_BLOCK PUBLIC FB_SetupCtrlAutoAdjust EXTENDS FB_SetupArmCtrlBase
VAR_INPUT
END_VAR
VAR_OUTPUT
END_VAR
VAR
END_VAR

METHOD PUBLIC init : BOOL
VAR_IN_OUT CONSTANT
	i_setupArm	:FB_SetupArm;
END_VAR
VAR_IN_OUT 
	r_setupArmCtrlCmd :ST_SetupArmCtrlCmds;
END_VAR
SUPER^.Init(i_setupArm,r_setupArmCtrlCmd);
END_METHOD

END_FUNCTION_BLOCK

// ---- FBs_SetupControllers/FB_SetupCtrlJnt3GraCali.TcPOU
// Brief: setup arm gravity calibration
// For trajectory synchronizaiton, the planner generate a trajecotry for setup joint3/5 and slave joint 1-3, but only former used here 
FUNCTION_BLOCK PUBLIC FB_SetupCtrlJnt3GraCali EXTENDS FB_SetupArmCtrlBase
VAR_INPUT
END_VAR
VAR_OUTPUT
END_VAR
VAR
// cali trajectory
	m_caliMotionSegs :INT :=3;
	m_graCaliTraj:ARRAY [1..3] OF LREAL:=[0.002,0.198,0.002];
	
	m_caliMaxjntVel:LREAL:=0.01;
	m_caliMaxjntAcc:LREAL:=0.5;
	m_caliMaxjntJerk:LREAL:=1.0;
	
	m_caliTrajIdx: INT := 1;
	m_caliPlanner: ARRAY[1..3] OF FB_BasicDoubleS;
	
END_VAR

// override this function in each exact controller
METHOD PROTECTED calcCmdJntPos : BOOL
VAR_IN_OUT CONSTANT
	i_setupArm	:FB_SetupArm;
END_VAR


VAR 
	i :INT;
	curJntVel :Vec5d;
END_VAR
// safety check
IF ABS(i_setupArm.curJntVel[3]) > 0.02 THEN
	m_isFinished:=TRUE;
	RETURN;
END_IF

// check if planner is ready
IF m_caliPlanner[m_caliTrajIdx].isGene = FALSE THEN
	calcCmdJntPos:=FALSE;
	RETURN;
END_IF

// traj plan
calcCmdJntPos :=m_caliPlanner[m_caliTrajIdx].evaluate(m_timePeriod, q=> m_cmdJntPos[3], q_dot=>m_cmdJntVel[3], q_ddot=> m_cmdJntAcc[3]);

// check if to transit to next segment
IF(m_timePeriod > m_caliPlanner[m_caliTrajIdx].duration  AND ABS(i_setupArm.curJntVel[3])<GVL_SlaveControlParameters.g_jntStaticVelThres) THEN
	m_caliTrajIdx:=m_caliTrajIdx+1;
	m_timePeriod:=0;
END_IF

// check if to terminated
IF(m_caliTrajIdx > m_caliMotionSegs) THEN
	m_isFinished:=TRUE;
END_IF
END_METHOD

METHOD PUBLIC init : BOOL
VAR_IN_OUT CONSTANT
	i_setupArm	:FB_SetupArm;
END_VAR
VAR_IN_OUT 
	r_setupArmCtrlCmd :ST_SetupArmCtrlCmds;
END_VAR

VAR
	i,j :INT;
	startJntPos,endJntPos :LREAL;
	q,v:ARRAY[1..2] OF lreal;
END_VAR
SUPER^.Init(i_setupArm,r_setupArmCtrlCmd);
m_jntEnableFlag[3]:=1;
m_jntOPMode[3]:= DriverOPMode_Pos;
m_caliTrajIdx :=1;

// traj plan
// fisrt segment
q[1]:=i_setupArm.curJntPos[3];
q[2]:=m_graCaliTraj[1];
v[1]:=0;
v[2]:=0;
m_caliPlanner[1].init(q,v,m_caliMaxjntVel, m_caliMaxJntAcc, m_caliMaxJntJerk);

// other segments
FOR i:=2 TO m_caliMotionSegs DO 
	q[1]:=m_graCaliTraj[i-1];
	q[2]:=m_graCaliTraj[i];
	m_caliPlanner[i].init(q,v,m_caliMaxjntVel, m_caliMaxJntAcc, m_caliMaxJntJerk);
END_FOR
END_METHOD

END_FUNCTION_BLOCK

// ---- FBs_SetupControllers/FB_SetupCtrlJnt5GraCali.TcPOU
// Brief: setup arm gravity calibration
// For trajectory synchronizaiton, the planner generate a trajecotry for setup joint3/5 and slave joint 1-3, but only former used here 
FUNCTION_BLOCK PUBLIC FB_SetupCtrlJnt5GraCali EXTENDS FB_SetupArmCtrlBase
VAR_INPUT
END_VAR
VAR_OUTPUT
END_VAR
VAR
// cali trajectory
	m_caliMotionSegs :INT :=3;
	m_graCaliTraj:ARRAY [1..3] OF LREAL:=[PI/2-pi/3, PI/2-PI/6, PI/2-pi/3];
	
		 
	m_caliMaxjntVel:LREAL:=2.5 * g_deg2Rad;
	m_caliMaxjntAcc:LREAL:=0.5;
	m_caliMaxjntJerk:LREAL:=2.0;
	
	m_caliTrajIdx: INT := 1;
	m_caliPlanner: ARRAY[1..3] OF FB_BasicDoubleS;
	
END_VAR

// override this function in each exact controller
METHOD PROTECTED calcCmdJntPos : BOOL
VAR_IN_OUT CONSTANT
	i_setupArm	:FB_SetupArm;
END_VAR


VAR 
	i :INT;
	curJntVel :Vec5d;
END_VAR
// safety check
IF ABS(i_setupArm.curJntVel[5]) > 0.25 THEN
	m_isFinished:=TRUE;
	RETURN;
END_IF

// check if planner is ready
IF m_caliPlanner[m_caliTrajIdx].isGene = FALSE THEN
	calcCmdJntPos:=FALSE;
	RETURN;
END_IF

// traj plan
calcCmdJntPos :=m_caliPlanner[m_caliTrajIdx].evaluate(m_timePeriod, q=> m_cmdJntPos[5], q_dot=>m_cmdJntVel[5], q_ddot=> m_cmdJntAcc[5]);

// check if to transit to next segment
IF(m_timePeriod > m_caliPlanner[m_caliTrajIdx].duration  AND ABS(i_setupArm.curJntVel[5])<GVL_SlaveControlParameters.g_jntStaticVelThres) THEN
	m_caliTrajIdx:=m_caliTrajIdx+1;
	m_timePeriod:=0;
END_IF

// check if to terminated
IF(m_caliTrajIdx > m_caliMotionSegs) THEN
	m_isFinished:=TRUE;
END_IF
END_METHOD

METHOD PUBLIC init : BOOL
VAR_IN_OUT CONSTANT
	i_setupArm	:FB_SetupArm;
END_VAR
VAR_IN_OUT 
	r_setupArmCtrlCmd :ST_SetupArmCtrlCmds;
END_VAR

VAR
	i,j :INT;
	startJntPos,endJntPos :LREAL;
	q,v:ARRAY[1..2] OF lreal;
END_VAR
SUPER^.Init(i_setupArm,r_setupArmCtrlCmd);
m_jntEnableFlag[5]:=1;
m_jntOPMode[5]:= DriverOPMode_PosTrq;
m_caliTrajIdx :=1;

// traj plan
// fisrt segment
q[1]:=i_setupArm.curJntPos[5];
q[2]:=m_graCaliTraj[1];
v[1]:=0;
v[2]:=0;
m_caliPlanner[1].init(q,v,m_caliMaxjntVel, m_caliMaxJntAcc, m_caliMaxJntJerk);

// other segments
FOR i:=2 TO m_caliMotionSegs DO 
	q[1]:=m_graCaliTraj[i-1];
	q[2]:=m_graCaliTraj[i];
	m_caliPlanner[i].init(q,v,m_caliMaxjntVel, m_caliMaxJntAcc, m_caliMaxJntJerk);
END_FOR
END_METHOD

END_FUNCTION_BLOCK

// ---- FBs_SetupControllers/FB_SetupCtrlDisable.TcPOU
// Brief: Setup Arm Error Hold
FUNCTION_BLOCK PUBLIC FB_SetupCtrlDisable EXTENDS FB_SetupArmCtrlBase
VAR_INPUT
END_VAR
VAR_OUTPUT
END_VAR
VAR
END_VAR

END_FUNCTION_BLOCK

// ---- FBs_SetupControllers/FB_SetupCtrlPerformance.TcPOU
FUNCTION_BLOCK FB_SetupCtrlPerformance EXTENDS FB_SetupArmCtrlBase
VAR_INPUT
END_VAR
VAR_OUTPUT
END_VAR
VAR CONSTANT
	//max number of data recording points
	m_dataSum:INT:=8000;
END_VAR

VAR
	//test step
	m_testStep:INT:=-1;
	
	//Extreme joint position
	m_minJntPos: ARRAY[1..g_setupJntNum] OF LREAL;
	m_maxJntPos: ARRAY[1..g_setupJntNum] OF LREAL;
	
	//home position
	m_homeJntPos:ARRAY[1..g_setupJntNum] OF LREAL;
	
	//arm parameters
	m_armId:INT;
	
	//index
	i,j,id,idx:INT;
	
	//trajectory planner
	m_caliTrajIdx: INT := 1;
	m_jntIdx:INT:=1;
	m_caliMotionSegs :INT :=4;
	m_caliPlanner: ARRAY[3..5,1..4] OF FB_setupTrajMoveJ;
	
	//trajectory velocity/acceleration/jerk
	m_caliMaxjntVel:Vec5d:=[2(1),0.01, 2(2.5*g_deg2Rad)];
	m_caliMaxjntAcc:Vec5d:=[2(1),0.5,2(0.5)];
	m_caliMaxjntJerk:Vec5d:=[2(1),1.0,2(2.0)];
		
	//sampling interval
	m_samplingInterval:INT:=80;
	
	//Number of data records
	m_dataRecordNum_2,m_dataRecordNum_3:ARRAY[1..g_setupJntNum] OF INT;
		
	//The current values of the second and third trajectories
	m_jntCurrentId2:ARRAY[1..m_dataSum,1..g_setupJntNum] OF LREAL;
	m_jntCurrentId3:ARRAY[1..m_dataSum,1..g_setupJntNum] OF LREAL;
	
	//friction record value
	m_CoulombFriction,m_ViscousFriction:ARRAY[1..m_dataSum,1..g_setupJntNum] OF LREAL;
	
	//friction summation
	m_CoulombFrictionSum,m_ViscousFrictionSum:ARRAY[1..g_setupJntNum] OF LREAL;
	
	//friction averange
	m_CoulombFrictionAve,m_ViscousFrictionAve:ARRAY[1..g_setupJntNum] OF LREAL;
	
	//friction maxmum value
	m_CoulombFrictionMax,m_ViscousFrictionMax:ARRAY[1..g_setupJntNum] OF LREAL;
	
	initJntPos,startJntPos,endJntPos :Vec5d;
END_VAR

// override this function in each exact controller
METHOD PROTECTED calcCmdJntPos : BOOL
VAR_IN_OUT CONSTANT
	i_setupArm	:FB_SetupArm;
END_VAR

CASE m_testStep OF 
	0: //test the motion range/joint friction/joint gap
		IF m_caliPlanner[m_jntIdx,m_caliTrajIdx].isGene = FALSE THEN
			calcCmdJntPos:=FALSE;
			RETURN;
		END_IF
		
		// traj plan
		calcCmdJntPos :=m_caliPlanner[m_jntIdx,m_caliTrajIdx].evaluate(m_timePeriod, jntPos=> m_cmdJntPos, jntVel=>m_cmdJntVel, jntAcc=> m_cmdJntAcc);
		
		// check if to transit to next segment		
		IF(m_timePeriod > m_caliPlanner[m_jntIdx,m_caliTrajIdx].duration) THEN
			m_caliTrajIdx:=m_caliTrajIdx+1;
			m_timePeriod:=0;
			idx:=0;
			id:=0;
			IF (m_caliTrajIdx>m_caliMotionSegs) THEN
				m_jntIdx:=m_jntIdx+1;
				m_caliTrajIdx:=1;				
			END_IF			
		END_IF
		
		//If all joints have been tested, enter the data processing flow
		IF (m_jntIdx>5) THEN
			m_testStep:=10;
		END_IF
		
		//Record the current value during the testing process
		IF (m_caliTrajIdx=2) THEN
			idx:=idx+1;
			IF (idx>=m_samplingInterval) THEN
				idx:=0;
				id:=id+1;
				m_dataRecordNum_2[m_jntIdx]:=id;
				m_jntCurrentId2[id,m_jntIdx]:=i_setupArm.filtJntCurrent[m_jntIdx]*GVL_SetupMotorParameters.g_motorDir[m_jntIdx];
			END_IF			
		ELSIF (m_caliTrajIdx=3) THEN
			idx:=idx+1;
			IF (idx>=m_samplingInterval) THEN
				idx:=0;
				id:=id+1;
				m_dataRecordNum_3[m_jntIdx]:=id;
				m_jntCurrentId3[id,m_jntIdx]:=i_setupArm.filtJntCurrent[m_jntIdx]*GVL_SetupMotorParameters.g_motorDir[m_jntIdx];
			END_IF			
		END_IF
		
		
	10: //Process the data from the above steps				
		FOR j:=3 TO 5 BY 1 DO
			id:=0;
			FOR i:=1 TO m_dataRecordNum_2[j] BY 1 DO 
				idx:=m_dataRecordNum_3[j]-i+1;
				IF (idx>0) THEN
					id:=id+1; //Number of groups for recording data
					m_CoulombFriction[i,j]:=(m_jntCurrentId2[i,j]-m_jntCurrentId3[idx,j])/2;
					m_ViscousFriction[i,j]:=(m_jntCurrentId2[i,j]+m_jntCurrentId3[idx,j])/2;
					
					m_CoulombFrictionSum[j]:=m_CoulombFrictionSum[j]+m_CoulombFriction[i,j];
					m_ViscousFrictionSum[j]:=m_ViscousFrictionSum[j]+m_ViscousFriction[i,j];
					
					IF (m_CoulombFriction[i,j]>m_CoulombFrictionMax[j]) THEN
						m_CoulombFrictionMax[j]:=m_CoulombFriction[i,j];
					END_IF
					
					IF (m_ViscousFriction[i,j]>m_ViscousFrictionMax[j]) THEN
						m_ViscousFrictionMax[j]:=m_ViscousFriction[i,j];
					END_IF				
				END_IF				
			END_FOR			
			//Calculate the mean of frictional force
			m_CoulombFrictionAve[j]:=m_CoulombFrictionSum[j]/id;
			m_ViscousFrictionAve[j]:=m_ViscousFrictionSum[j]/id;			
		END_FOR
		
		m_testStep:=-1;
		m_isFinished:=TRUE;
		
		
	20: //
		
		
	-1: //
END_CASE
END_METHOD

// override this function in each exact controller
// NOTICE: set joint control mode here, and do some initialization if needed
METHOD PUBLIC init : BOOL
VAR_IN_OUT CONSTANT
	i_setupArm	:FB_SetupArm;
END_VAR
VAR_IN_OUT 
	r_setupArmCtrlCmd :ST_SetupArmCtrlCmds;
END_VAR
VAR
	//joint position variables
	//initJntPos,startJntPos,endJntPos :Vec5d;
END_VAR
SUPER^.Init(i_setupArm,r_setupArmCtrlCmd);
m_jntEnableFlag:=g_onesVec5i; m_jntEnableFlag[1]:=0; m_jntEnableFlag[2]:=0;
m_jntOPMode:= g_setupAllPosMode;


//arm id and joint position initial
m_armId:=i_setupArm.armIdx;
initJntPos:=i_setupArm.curJntPos;
startJntPos:=initJntPos;
endJntPos:=initJntPos;


//Assignment of joint position limit values and home position
FOR j:=1 TO g_setupJntNum BY 1 DO
	m_minJntPos[j]:=GVL_SetupMotorParameters.g_minJntPos[m_armId,j];
	m_maxJntPos[j]:=GVL_SetupMotorParameters.g_maxJntPos[m_armId,j];
	m_homeJntPos[j]:=(m_minJntPos[j]+m_maxJntPos[j])/2;
END_FOR


//step/joint id/ trajectory id
m_testStep:=0;
m_caliTrajIdx :=1;
m_jntIdx:=3;


//Trajectory generator initialization
FOR j:=3 TO 5 BY 1 DO
	FOR id:=1 TO 4 BY 1 DO
		startJntPos:=endJntPos;
		endJntPos:=m_homeJntPos;
		
		IF (id=1) THEN
			endJntPos[j]:=m_minJntPos[j]; //minimum
		ELSIF (id=2) THEN
			endJntPos[j]:=m_maxJntPos[j]; //maximum
		ELSIF (id=3) THEN
			endJntPos[j]:=m_minJntPos[j]; //minimum
		ELSIF (id=4) THEN
			endJntPos[j]:=m_homeJntPos[j]; //home
		END_IF		
		m_caliPlanner[j,id].init(startJntPos,endJntPos,m_caliMaxjntVel, m_caliMaxJntAcc, m_caliMaxJntJerk);
	END_FOR
END_FOR


//Initialization of calculation results
FOR j:=1 TO g_setupJntNum BY 1 DO
	m_CoulombFrictionSum[j]:=0; 	m_CoulombFrictionMax[j]:=0; 	m_CoulombFrictionAve[j]:=0;	
	m_ViscousFrictionSum[j]:=0;	 m_ViscousFrictionMax[j]:=0;	 m_ViscousFrictionAve[j]:=0;
END_FOR
END_METHOD

END_FUNCTION_BLOCK

// ---- Mains/RobotDynamics.TcPOU
PROGRAM RobotDynamics

VAR
	// slave robot arms joint data
	m_slaveJointsData AT %I* :ST_SlaveJointData;
	
	// setup joint5 position
	m_setupJointData AT %I* :ST_SetupJointData;
	
	// instrument info
	m_instruInfo AT %I* :ARRAY[1..g_sArmNum] OF ST_InstruStatus;
	
	// dynamic output
	m_slaveDynaData AT %Q* : ST_SlaveDynaData;
	m_setupJnt3Gravity AT %Q* : ARRAY[1..g_sArmNum] OF LREAL;
	m_setupJnt5Gravity AT %Q* : ARRAY[1..g_sArmNum] OF LREAL;
	
	// flag to init robot dynamic model
	m_robotDynaInit :BOOL :=FALSE;
	
	// grivity model block
	m_slaveGravityModel :ARRAY[1..g_sArmNum] OF FB_SlaveGravity;
	m_setupGravityModel :ARRAY[1..g_sArmNum] OF FB_SetupGravity;
	
	// slave dynamic block
	m_slaveDynamicModel :ARRAY[1..g_sArmNum] OF FB_SlaveDynamic;
	
	// instument out-of-view check
	m_instruViewCheck :FB_InstruViewCheck;

	// code execute time measure
	m_codeTime : Profiler;
	
	// tmp variables
	i: INT;
	
END_VAR

m_codeTime(START:=TRUE, RESET:=TRUE);

// robot dynamic model init
IF m_robotDynaInit =FALSE THEN
	FOR i:=1 TO g_sArmNum DO
		m_slaveGravityModel[i].Init(i);
		m_setupGravityModel[i].init(i);
		m_slaveDynamicModel[i].init(i);
	END_FOR
	m_instruViewCheck.init();

	m_robotDynaInit:=TRUE;
END_IF


FOR i:=1 TO g_sArmNum DO
	// run gravity model
	m_slaveDynaData.m_gravity[i]:=m_slaveGravityModel[i].run(m_setupJointData.m_curJntPos[i][5], m_slaveJointsData.m_curJntPos[i],m_instruInfo[i]);
	m_setupGravityModel[i].run(m_setupJointData.m_curJntPos[i], m_slaveJointsData.m_curJntPos[i],m_instruInfo[i], o_jnt3Gravity=> m_setupJnt3Gravity[i], o_jnt5Gravity=> m_setupJnt5Gravity[i]);
	
	// run dynamic model
	m_slaveDynamicModel[i].updateDynamic(m_slaveJointsData.m_curJntPos[i]);
	m_slaveDynaData.m_massMat[i]:= m_slaveDynamicModel[i].jntMassMat;
END_FOR

m_instruViewCheck.run(m_setupJointData.m_curJntPos, m_slaveJointsData.m_curDHJntPos, m_instruInfo);
m_slaveDynaData.m_insruViewData:=m_instruViewCheck.m_instruImgBoundPos;


m_codeTime(START:=FALSE);

END_PROGRAM

// ---- Sandbox/FB_SlaveArmCheck.TcPOU
FUNCTION_BLOCK FB_SlaveArmCheck
VAR_INPUT
END_VAR
VAR_OUTPUT
END_VAR
VAR
	// final arm/joint error flag
	m_armErrFlag :ARRAY[1..g_sArmNum] OF BOOL:=[4(FALSE)];
	m_jntErrFlag :ARRAY[1..g_sArmNum] OF Vec8b;
	
	// cartesian pose error flag
	m_cartPoseErrFlag :ARRAY[1..g_sArmNum] OF BOOL;
	m_cartPoseErrCounts:ARRAY[1..g_sArmNum] OF INT;
	m_cartPosErr :ARRAY[1..g_sArmNum] OF Vec3d;	// cartesian position error
	m_cartOriErr:ARRAY[1..g_sArmNum] OF  Vec3d;	// cartesian rotation angle (angle  * axis)
	
	// joint control error flag
	m_jntCtrlErrFlag :ARRAY[1..g_sArmNum] OF Vec8b;
	m_jntCtrlErrCounts :ARRAY[1..g_sArmNum] OF Vec8i;
	m_jntCtrlErr:ARRAY[1..g_sArmNum]  OF Vec8d;		// joint position control error
	
	// joint encoder error flag
	m_jntEncErrFlag :ARRAY[1..g_sArmNum] OF Vec8b;
	m_jntEncErrCounts :ARRAY[1..g_sArmNum] OF Vec8i ;
	m_jntEncErr:ARRAY[1..g_sArmNum]  OF Vec8d;		// motor and joint encoder error
	
	// joint velocity error flag
	m_jntVelErrFlag :ARRAY[1..g_sArmNum] OF Vec8b;
	m_jntVelErrCounts :ARRAY[1..g_sArmNum] OF Vec8i;
	
	// joint position limit error flag
	m_jntLimitErrFlag :ARRAY[1..g_sArmNum] OF Vec8b;
	m_jntLimitErrCounts :ARRAY[1..g_sArmNum] OF Vec8i;

END_VAR

METHOD check : BOOL
VAR_IN_OUT CONSTANT
	i_slaveStatus : ST_SlaveStatus;
	i_slaveJointData :ST_SlaveJointData;
END_VAR
VAR_OUTPUT
	o_errorFlag :ARRAY[1..g_sArmNum] OF BOOL ;
END_VAR

VAR
	i ,j:INT ;
END_VAR
// calculate error
FOR i:=1 TO g_sArmNum DO 
	// stop check if arm is already in error state
	IF m_armErrFlag[i] OR i_slaveStatus.m_armState[i]=SlaveArmState_Error OR i_slaveStatus.m_armState[i]=SlaveArmState_Disable THEN 
		CONTINUE;
	END_IF
	
	// only check cartesion pose error in master-slave mode within joint limit
	m_cartPoseErrFlag[i]:=FALSE;
	IF  SlaveArmState_MasterSlave = i_slaveStatus.m_armState[i] AND norm(i_slaveStatus.m_masterSlavePoseError[i])<g_smallNum THEN 
		m_cartPoseErrFlag[i]:=poseErrCheck(i_slaveStatus.m_cmdArmPose[i],  i_slaveStatus.m_simArmPose[i],
											m_cartPoseErrCounts[i], m_cartPosErr[i], m_cartOriErr[i]);
	END_IF
	
	// joint control error
	m_jntCtrlErrFlag[i]:=jntCtrlErrCheck(i_slaveJointData.m_cmdJntPos[i], i_slaveJointData.m_curJntPos[i],
										m_jntCtrlErrCounts[i], m_jntCtrlErr[i]);
	
	// encoder error
	m_jntEncErrFlag[i]:=jntEncErrCheck(i_slaveJointData.m_curMotorPos[i], i_slaveJointData.m_curLinkPos[i],
										m_jntEncErrCounts[i], m_jntEncErr[i]);
										
	// joint limit error
	m_jntLimitErrFlag[i]:=jntLimitErrCheck(i_slaveJointData.m_curJntPos[i],m_jntLimitErrCounts[i]);
										
	// final arm error status check
	IF  m_cartPoseErrFlag[i] THEN
		m_armErrFlag[i]:=TRUE;
		CONTINUE;
	END_IF
	
	FOR j:=1 TO g_sJntNum DO 
		m_jntErrFlag[i] := g_zeroVec8b;
		IF m_jntCtrlErrFlag[i][j] OR m_jntEncErrFlag[i][j] OR m_jntVelErrFlag[i][j] OR m_jntLimitErrFlag[i][j] THEN
			m_jntErrFlag[i][j] := TRUE;
			m_armErrFlag[i]:=TRUE;
		END_IF
	END_FOR
	
END_FOR

o_errorFlag:=m_armErrFlag;
END_METHOD

METHOD jntCtrlErrCheck : Vec8b
VAR_INput
	i_cmdJntPos : Vec8d;
	i_curJntPos : Vec8d;
END_VAR
VAR_IN_OUT
	r_errCount:Vec8i;
	r_jntCtrlErr :Vec8d;
END_VAR

VAR
	i :INT;
	err:Vec8d;
END_VAR
vecSub(i_cmdJntPos,i_curJntPos,  err);
r_jntCtrlErr:=err;

// joint error check
//NOTE: only check the first three joints.
FOR i:=1 TO 3 DO 
	IF  ABS(r_jntCtrlErr[i]) > g_slaveMaxJntCtrlErr[i] THEN
		r_errCount[i]:=r_errCount[i]+1;
	ELSE
		r_errCount[i] :=0;	
	END_IF
	jntCtrlErrCheck[i]:= r_errCount[i]>=g_faultTriggerCountsLarge;
END_FOR
END_METHOD

METHOD jntEncErrCheck : Vec8b
VAR_INput
	i_motorJntPos : Vec8d;
	i_linkJntPos : Vec8d;
END_VAR
VAR_IN_OUT
	r_errCount:Vec8i;
	r_jntEncErr :Vec8d;
END_VAR

VAR
	i :INT;
	err:Vec8d;
END_VAR
vecSub(i_motorJntPos,i_linkJntPos,  err);
r_jntEncErr:=err;

// joint error check
FOR i:=1 TO g_sJntNum DO 
	IF  ABS(r_jntEncErr[i]) > g_slaveMaxJntCtrlErr[i] THEN
		r_errCount[i]:=r_errCount[i]+1;
	ELSE
		r_errCount[i] :=0;
	END_IF
	jntEncErrCheck[i]:= r_errCount[i]>=g_faultTriggerCounts;
END_FOR

// NOTE: power box joints are easy to trigger encoder error during instrument mount, so this part is diabled now
FOR i:=4 TO g_sJntNum DO
	jntEncErrCheck[i] := false;
END_FOR
END_METHOD

METHOD jntLimitErrCheck : Vec8b
VAR_INput
	i_curJntPos : Vec8d;
END_VAR
VAR_IN_OUT
	r_errCount:Vec8i;
END_VAR

VAR
	i :INT;
END_VAR
// joint limit check
//NOTE: only check the first three joints.
FOR i:=1 TO 3 DO 
	IF  i_curJntPos[i] > GVL_SlaveMotorParameters.g_maxJntPos[i] + g_slaveJntPosLimitBuffer[i] OR
		i_curJntPos[i] < GVL_SlaveMotorParameters.g_minJntPos[i] - g_slaveJntPosLimitBuffer[i] THEN
		r_errCount[i]:=r_errCount[i]+1;
	ELSE
		r_errCount[i] :=0;	
	END_IF
	jntLimitErrCheck[i]:= r_errCount[i]>=g_faultTriggerCounts;
END_FOR
END_METHOD

METHOD poseErrCheck : BOOL
VAR_INPUT
	i_cmdPose : ST_Frame;
	i_curPose :ST_Frame;
END_VAR
VAR_IN_OUT
	r_errCount:INT;
	r_posErr :Vec3d;
	r_oriErr :Vec3d;
END_VAR

VAR
	posErr,oriErr:Vec3d;
	matT,rotErr:Mat3d;
	errAngle :LREAL;
	errAxis :Vec3d;
END_VAR
vecSub(i_cmdPose.m_pos, i_curPose.m_pos,posErr);
r_posErr:=posErr;

matTranspose(i_cmdPose.m_rot, matT);
matMultiply(matT,i_curPose.m_rot, rotErr);
rot2AngAxis(rotErr, angle=>errAngle, axis=>errAxis);
vecMultiNum(errAxis, errAngle,oriErr);
r_oriErr:=oriErr;
	
IF  norm(posErr)>g_maxCartPosErr OR norm(oriErr)> g_maxCartOriErr THEN
	r_errCount:= r_errCount +1;
ELSE 
	r_errCount:=0;
END_IF
poseErrCheck:= r_errCount >= g_faultTriggerCountsLarge;
END_METHOD

END_FUNCTION_BLOCK

// ---- Sandbox/FB_SlaveCtrlAdjust_bak1.TcPOU
// Brief: Slave Arm Adjust
FUNCTION_BLOCK PUBLIC FB_SlaveCtrlAdjust_bak1 EXTENDS FB_SlaveArmCtrlBase
VAR
	// velocity for full damping
	m_maxAdjustVel :Vec3d := [1.2, 1.2, 0.3];
	
	// velocity start to enable damping
	m_velLBForDamp :Vec3d := [1.0, 1.0, 0.2];
	
	// max damp
	m_maxDamp :Vec3d := [50, 50, 500];
	
	// distance buffer from joint limit to start damp
	m_limitBufferForDamp :Vec3d :=[20*g_deg2Rad, 20*g_deg2Rad, 0.03];
	
	//limit protect method selection
	m_methodSelect:INT:=2;
	
	//reverse motion enable flag
	m_reverseMotionEnable:ARRAY[1..3] OF BOOL;
	
	//hard Limit position---[minVal,maxVal]
	m_hardLimit:ARRAY[1..3,1..2] OF LREAL;
	
	//soft Limit position---[minVal,maxVal]
	m_softLimit:ARRAY[1..3,1..2] OF LREAL;
	
	//damp force start position
	m_dampStartPos:ARRAY[1..3,1..2] OF LREAL;
	
	//distance from hard limit position to soft limit position
	m_distHard2Soft:Vec3d := [20*g_deg2Rad, 20*g_deg2Rad, 0.03];
	
	//distance from start position to soft limit position
	m_distStart2Soft:Vec3d := [20*g_deg2Rad, 20*g_deg2Rad, 0.03];
	
	//Extreme speed point--- [startPosVel,softPosVel,hardPosVels
	m_limitVelocity:ARRAY[1..3,1..3] OF LREAL:=[1.0,0.2,-0.2,   1.0,0.2,-0.2,   0.2,0,-0.2];
	
	//position array
	m_posArr:ARRAY[1..3,1..6] OF LREAL;
	
	//velocity array
	m_velArr:ARRAY[1..3,1..6] OF LREAL;
	
	//velocity difference
	m_velDiff:Vec3d;
	
	//speed setpoint
	m_speedPoint:Vec3d;
	
	//damping factor
	m_dampFactor:Vec3d:= [50, 50, 100];
	
	//flag if joint add damp force
	m_ifAddDamp:ARRAY[1..3] OF BOOL;
END_VAR

// override this function in each exact controller
METHOD PROTECTED calcCmdJntPos : BOOL
VAR_IN_OUT CONSTANT
	i_endoscopePose : ST_Frame;
	i_masterStatus :ST_MasterStatus;
	i_setupStatus: ST_SetupStatus;
	i_slaveArm :FB_SlaveArm;
END_VAR
m_cmdJntPos[1]:=i_slaveArm.curJntPos[1];
m_cmdJntPos[2]:=i_slaveArm.curJntPos[2];
m_cmdJntPos[3]:=i_slaveArm.curJntPos[3];
IF m_jntOPMode[8] = DriverOPMode_Trq THEN
	m_cmdJntPos[8]:=i_slaveArm.curJntPos[8];
END_IF
IF m_jntOPMode[7] = DriverOPMode_Trq THEN
	m_cmdJntPos[7]:=i_slaveArm.curJntPos[7];
END_IF

m_cmdCartPose:=i_slaveArm.curCartPose;
END_METHOD

// override this function in each exact controller
METHOD PROTECTED calcCmdJntTrq : BOOL
VAR_IN_OUT CONSTANT
	i_endoscopePose : ST_Frame;
	i_masterStatus :ST_MasterStatus;
	i_setupStatus: ST_SetupStatus;
	i_slaveArm :FB_SlaveArm;
END_VAR
VAR
	i :INT;
	dampScale :LREAL;
	limitDis:LREAL;
END_VAR
// set joint torque to zero in default
m_cmdJntTrq := g_zeroVec8d;

// enable endoscope rotation joint if external torque exceed specific value
IF i_slaveArm.instrument.onChipData.m_InstruReadSucceed AND i_slaveArm.instrument.instruType = InstruType_Endoscope AND ABS(i_slaveArm.filtJntCurrent[8]) > 100 THEN
		m_jntOPMode[8]:=DriverOPMode_Trq;
END_IF


// add damp near joint limit
IF (m_methodSelect=1) THEN
	FOR i:=1 TO 3 DO
		IF (i_slaveArm.curJntPos[i] > GVL_SlaveMotorParameters.g_maxDHJntPos[i] - m_limitBufferForDamp[i] AND  i_slaveArm.curJntVel[i]> 0 ) 
			OR (i_slaveArm.curJntPos[i] < GVL_SlaveMotorParameters.g_minDHJntPos[i] + m_limitBufferForDamp[i] AND  i_slaveArm.curJntVel[i]<0 )  THEN
			limitDis := MIN(GVL_SlaveMotorParameters.g_maxDHJntPos[i] - i_slaveArm.curJntPos[i], i_slaveArm.curJntPos[i]-GVL_SlaveMotorParameters.g_minDHJntPos[i]);
			dampScale  :=LIMIT(0, 1-limitDis/m_limitBufferForDamp[i],1);
			m_cmdJntTrq[i]:= -dampScale * m_maxDamp[i] * i_slaveArm.curJntVel[i];
		END_IF	
	END_FOR
END_IF


//enabel accidental movement
FOR i:=1 TO 3 BY 1 DO
	IF (m_reverseMotionEnable[i]=FALSE) AND ((i_slaveArm.curJntPos[i]>m_posArr[i,5]) AND (i_slaveArm.curJntPos[i]<m_posArr[i,2])) THEN
		m_reverseMotionEnable[i]:=TRUE;
		m_velArr[i,3]:=m_limitVelocity[i,3];
		m_velArr[i,6]:=-m_limitVelocity[i,3];
	END_IF
END_FOR


//Calculate the limit value of speed
IF (m_methodSelect=2) THEN
	calcSpeedSetPoint(i_slaveArm:= i_slaveArm);
	FOR i:=1 TO 3 DO
		IF (m_ifAddDamp[i]=TRUE)THEN
			m_velDiff[i]:=m_speedPoint[i]-i_slaveArm.curJntVel[i];
			m_cmdJntTrq[i]:=m_dampFactor[i]*m_velDiff[i];
		ELSE
			m_velDiff[i]:=0;
			m_cmdJntTrq[i]:=0;
		END_IF		
	END_FOR
END_IF


// compute damp
FOR i:=1 TO 3 DO
	IF ABS(i_slaveArm.curJntVel[i]) > m_velLBForDamp[i] THEN 
		dampScale:=LIMIT(0, (ABS(i_slaveArm.curJntVel[i])- m_velLBForDamp[i])/(m_maxAdjustVel[i] - m_velLBForDamp[i]), 1 );
		m_cmdJntTrq[i] :=m_cmdJntTrq[i] -i_slaveArm.curJntVel[i] * m_maxDamp[i] * dampScale;
	END_IF
END_FOR
END_METHOD

METHOD calcSpeedSetPoint : BOOL
VAR_INPUT
	i_slaveArm :FB_SlaveArm;
END_VAR

VAR
	i:INT;
END_VAR

//Calculate the limit value of speed
FOR i:=1 TO 3 DO
	IF (i_slaveArm.curJntPos[i]>m_posArr[i,2]) THEN
		linearInterpolation(i_x1:= m_posArr[i,2], i_y1:= m_velArr[i,2], i_x2:= m_posArr[i,3], i_y2:= m_velArr[i,3], i_x:= i_slaveArm.curJntPos[i], o_y=> m_speedPoint[i]);
		IF (i_slaveArm.curJntVel[i]>m_speedPoint[i]) THEN
			m_ifAddDamp[i]:=TRUE;
		ELSE
			m_ifAddDamp[i]:=FALSE;
		END_IF		
		
	ELSIF (i_slaveArm.curJntPos[i]>m_posArr[i,1]) AND (i_slaveArm.curJntPos[i]<m_posArr[i,2]) THEN
		linearInterpolation(i_x1:= m_posArr[i,1], i_y1:= m_velArr[i,1], i_x2:= m_posArr[i,2], i_y2:= m_velArr[i,2], i_x:= i_slaveArm.curJntPos[i], o_y=> m_speedPoint[i]);
		IF (i_slaveArm.curJntVel[i]>m_speedPoint[i]) THEN
			m_ifAddDamp[i]:=TRUE;
		ELSE
			m_ifAddDamp[i]:=FALSE;
		END_IF	
		
	ELSIF (i_slaveArm.curJntPos[i]>m_posArr[i,5]) AND (i_slaveArm.curJntPos[i]<m_posArr[i,4]) THEN
		linearInterpolation(i_x1:= m_posArr[i,5], i_y1:= m_velArr[i,5], i_x2:= m_posArr[i,4], i_y2:= m_velArr[i,4], i_x:= i_slaveArm.curJntPos[i], o_y=> m_speedPoint[i]);
		IF (i_slaveArm.curJntVel[i]< m_speedPoint[i]) THEN
			m_ifAddDamp[i]:=TRUE;
		ELSE
			m_ifAddDamp[i]:=FALSE;
		END_IF
		
	ELSIF (i_slaveArm.curJntPos[i]<m_posArr[i,5]) THEN
		linearInterpolation(i_x1:= m_posArr[i,5], i_y1:= m_velArr[i,5], i_x2:= m_posArr[i,6], i_y2:= m_velArr[i,6], i_x:= i_slaveArm.curJntPos[i], o_y=> m_speedPoint[i]);
		IF (i_slaveArm.curJntVel[i]< m_speedPoint[i]) THEN
			m_ifAddDamp[i]:=TRUE;
		ELSE
			m_ifAddDamp[i]:=FALSE;
		END_IF
		
	ELSE
		m_speedPoint[i]:=0;
		m_ifAddDamp[i]:=FALSE;
	END_IF
END_FOR
END_METHOD

METHOD PUBLIC init : BOOL
VAR_IN_OUT CONSTANT
	i_slaveArm	:FB_SlaveArm;
END_VAR
VAR_IN_OUT 
	r_slaveArmCtrlCmd :ST_SlaveArmCtrlCmds;
END_VAR
VAR
	i :INT;
END_VAR
// check if to hold the command joint position unchanged
m_holdLastCmds := checkToHoldLastCmds(i_slaveArm);

//init
SUPER^.Init(i_slaveArm,r_slaveArmCtrlCmd);

// disable joints if this joint is an unrecoverable failure
FOR i:=1 TO g_sJntNum DO
	IF SafetyCheck.m_SafetyCheck.m_jntErrFlag[i_slaveArm.armIdx, 0, 3] OR  SafetyCheck.m_SafetyCheck.m_jntErrFlag[i_slaveArm.armIdx, i+g_setupJntNum, 3] THEN
		m_jntEnableFlag[i] := 0;
	ELSE
		m_jntEnableFlag[i] := 1;
	END_IF
END_FOR

// joint 1/2/3/7 run in torque mode
m_jntOPMode[1]:=DriverOPMode_Trq;
m_jntOPMode[2]:=DriverOPMode_Trq;
m_jntOPMode[3]:=DriverOPMode_Trq;
m_jntOPMode[4]:=DriverOPMode_PosTrq;
m_jntOPMode[5]:=DriverOPMode_PosTrq;
m_jntOPMode[6]:=DriverOPMode_PosTrq;
m_jntOPMode[7]:=DriverOPMode_PosTrq;
m_jntOPMode[8]:=DriverOPMode_PosTrq;

IF i_slaveArm.instrument.onChipData.m_InstruReadSucceed THEN
	IF i_slaveArm.instrument.instruType <> InstruType_Endoscope THEN
		m_jntOPMode[7]:=DriverOPMode_Trq;
	END_IF
END_IF

FOR i:=1 TO 3 DO
	//Set the lower limit value of the position
	m_hardLimit[i,1]:=GVL_SlaveMotorParameters.g_minDHJntPos[i];
	m_softLimit[i,1]:=m_hardLimit[i,1]+m_distHard2Soft[i];
	m_dampStartPos[i,1]:=m_softLimit[i,1]+m_distStart2Soft[i];
	
	//Set the upper limit value of the position
	m_hardLimit[i,2]:=GVL_SlaveMotorParameters.g_maxDHJntPos[i];	
	m_softLimit[i,2]:=m_hardLimit[i,2]-m_distHard2Soft[i];	
	m_dampStartPos[i,2]:=m_softLimit[i,2]-m_distStart2Soft[i];
	
	//position array
	m_posArr[i,1]:=m_dampStartPos[i,2]; m_posArr[i,2]:=m_softLimit[i,2]; m_posArr[i,3]:=m_hardLimit[i,2];
	m_posArr[i,4]:=m_dampStartPos[i,1]; m_posArr[i,5]:=m_softLimit[i,1]; m_posArr[i,6]:=m_hardLimit[i,1];
	
	//velocity array
	m_velArr[i,1]:=m_limitVelocity[i,1]; m_velArr[i,2]:=m_limitVelocity[i,2]; m_velArr[i,3]:=m_limitVelocity[i,3];
	m_velArr[i,4]:=-m_limitVelocity[i,1]; m_velArr[i,5]:=-m_limitVelocity[i,2]; m_velArr[i,6]:=-m_limitVelocity[i,3];
	
	//prevent accidental movement
	IF (i_slaveArm.curJntPos[i]>m_posArr[i,2]) OR (i_slaveArm.curJntPos[i]<m_posArr[i,5]) THEN
		m_reverseMotionEnable[i]:=FALSE;
		m_velArr[i,3]:=0;
		m_velArr[i,6]:=0;
	ELSE
		m_reverseMotionEnable[i]:=TRUE;
		m_velArr[i,3]:=m_limitVelocity[i,3];
		m_velArr[i,6]:=-m_limitVelocity[i,3];
	END_IF
END_FOR

IF (i_slaveArm.armIdx=1) OR (i_slaveArm.armIdx=2) THEN
	m_methodSelect:=1;
ELSE
	m_methodSelect:=2;
END_IF

// update commands to arm
copyCmds(r_slaveArmCtrlCmd);
END_METHOD

METHOD linearInterpolation : BOOL
VAR_INPUT
	i_x1:LREAL;
	i_y1:LREAL;
	i_x2:LREAL;
	i_y2:LREAL;
	i_x:LREAL;
END_VAR

VAR_OUTPUT
	o_y:LREAL;
END_VAR

VAR
	k:LREAL;
END_VAR

k:=(i_y2-i_y1)/(i_x2-i_x1);
o_y:=i_y1+k*(i_x-i_x1);
END_METHOD

END_FUNCTION_BLOCK

// ---- Sandbox/FB_SlaveCtrlMasterSlave_bak1.TcPOU
// Brief: Slave Arm MasterSlave controller
FUNCTION_BLOCK PUBLIC FB_SlaveCtrlMasterSlave_bak1 EXTENDS FB_SlaveArmCtrlBase
VAR_INPUT
END_VAR
VAR_OUTPUT
END_VAR
VAR
	// minimum distance between instrument tip and remote center
	m_minInstruRCDis:LREAL := 0.05;
	
	// master-slave motion scale
	m_MSMotionScale :LREAL;
		
	// gripper match angle threshold
	m_gripperMatchAngThres :LREAL := 2*g_deg2Rad;
	
	// control error thershold from joint limit back to free space
	m_maxPosTrackErr :LREAL := 0.05;
	m_maxOriTrackErr :LREAL :=g_deg2Rad * 5;
	
	// filter cut-off frequency for master-slave control
	m_macroCmdJntPosLpfCutoffFreq : LREAL :=5;
	m_microCmdJntPosLpfCutoffFreq : LREAL :=15;
	
	// last command joint position
	m_lastCmdJntPos :Vec8d;
	
	// simulated DH joint position
	m_simDHJntPos : Vec6d;
	
	// simulated slave twist of DH joint
	m_simDHJointVel :Vec6d;
		
	// enter master-slave control for the first time
	m_firstIn :BOOL := TRUE;
	
	// flag if reach joint limit
	m_reachMacroJntLimit :BOOL;
	m_reachWristJntLimit :BOOL;
	
	// master/slave origin pose when first enter master-slave control
	m_masterOriginPose : ST_Frame;
	m_slaveOriginPose : ST_Frame;
	
	// orientation deviation(in master coordinate) between master and slave when first enter control
	m_MSOriDeviation : Mat3d;
	
	// command joint position filter
	m_cmdJntPosLpf:ARRAY[1..8] OF FB_LowPassFilter;
	
	// commmand yaw angle and velocity
	m_cmdYawAngle :LREAL;
	m_cmdYawVel :LREAL;
	
	// comand yaw angle and velocity filter
	m_cmdYawAngLpf : FB_LowPassFilter;
	m_cmdYawVelLpf : FB_LowPassFilter;
	
	// master pose/velocity in monitor coordinate
	m_masterPose :ST_Frame;
	m_masterTwist : Vec6d;
	
	// master grip angle
	m_masterGripAngle : LREAL;
	
	// slave command/current pose in endoscope coordinate
	m_slaveCmdPoseInScope :ST_Frame;
	m_slavePoseInScope : ST_Frame;
	
	// slave command/current pose in cart
	m_slaveCmdPoseInCart :ST_Frame;
	m_slavePoseInCart : ST_Frame;
	
	// instrument controller
	m_basicInstruController : FB_BasicInstruControl;
	m_usKnifeController : FB_UltrosonicKnifeControl;
	
	// slave command grip angle and grip force level
	m_slaveCmdGripAngle :LREAL;
	m_slaveCmdGripForceLevel:LREAL;
	
	// slave pose error
	m_slavePosErr :Vec3d;
	m_slaveRotErr :Mat3d;
	m_errAngle : LREAL;
	m_errAxisLocal, m_errAxis :Vec3d;
	m_masterSlavePoseError :Vec6d;
	
	// velocity for slave to track master motion
	m_slaveTrackTwist :Vec6d;
	m_slaveCmdVel, m_slaveCmdWVel : Vec3d;
	
	// last master gripper angle
	m_lastMasterGripAngle :LREAL;
	
	// master gripper angle velocity
	m_masterGripAngleVel :LREAL;
	m_masterGripAngleVelLpf :FB_LowPassFilter;
	
	// flag to start gripper control
	m_gripperCtrlFlag :BOOL;
	
	// code execute time measure
	m_codeTime : Profiler;
	
END_VAR

METHOD PROTECTED calcCmdJntPos : BOOL
VAR_IN_OUT CONSTANT
	i_endoscopePose : ST_Frame;
	i_masterStatus :ST_MasterStatus;
	i_setupStatus: ST_SetupStatus;
	i_slaveArm :FB_SlaveArm;
END_VAR

VAR 
	i,j : INT;
	tmpMat3d : Mat3d;
	masterMotionRange : Vec3d;
	
	masterVelInScope, masterWVelInScope :Vec3d;
	masterVelInCart, masterWVelInCart :Vec3d;

	cmdVelScale :LREAL;
	invJaco :Mat6d;
	DHJntCmdDeltaPos :Vec6d;
	armJntJaco,armJntJacoInv, wristJntJaco :Mat3d;
	velByWristJnt,velByArmJnt : Vec3d;
	armDHJntVel, wristDHJntVel :Vec3d;
	tmpFrame : ST_Frame;
	slaveSimDHJntPos :Vec6d;
	jnt3Limit :LREAL;
END_VAR
m_codeTime(START:=TRUE, RESET:=TRUE);

IF isFinished THEN
	RETURN;
END_IF

// decide matched master arm index
FOR i:=1 TO g_mArmNum DO 
	IF i_masterStatus.m_teleSlaveArmIdx[i] = i_slaveArm.armIdx THEN
		m_masterPose := i_masterStatus.m_curArmPose[i];
		m_masterTwist := i_masterStatus.m_curArmTwist[i];
		m_masterGripAngle := i_masterStatus.m_gripAngle[i];
	END_IF
END_FOR

// compute slave pose in endoscope coordinate
m_slavePoseInCart := transform(i_setupStatus.m_curEndPose[i_slaveArm.armIdx], i_slaveArm.simCartPose);
tmpFrame :=invFrame(i_endoscopePose);
m_slavePoseInScope := transform(tmpFrame, m_slavePoseInCart);

// handle for the first time in
IF TRUE = m_firstIn THEN
	m_firstIn := FALSE;
	m_masterOriginPose :=m_masterPose;
	m_slaveOriginPose := m_slavePoseInScope;
	matTranspose(m_masterOriginPose.m_rot, tmpMat3d);
	matMultiply(tmpMat3d, m_slavePoseInScope.m_rot,m_MSOriDeviation);
	m_lastMasterGripAngle := m_masterGripAngle;
	
	// only update motion scale while entering teleControl 
	m_MSMotionScale := 1.0/ MAX(1,  i_masterStatus.m_motionScale);
END_IF

// compute master twist in slave arm coordinate
(*FOR i:=1 TO 3 DO
	masterVelInScope[i] := m_masterTwist[i]*i_masterStatus.m_motionScale;
	masterWVelInScope[i] := m_masterTwist[i+3];
END_FOR
matMultiVec(i_endoScopePose.m_rot, masterVelInScope, masterVelInCart);
matMultiVec(i_endoScopePose.m_rot, masterWVelInScope, masterWVelInCart);
matTranspose(i_setupStatus.m_curEndPose[i_slaveArm.armIdx].m_rot, tmpMat3d);
matMultiVec(tmpMat3d,masterVelInCart, m_masterFFVel);
matMultiVec(tmpMat3d,masterWVelInCart, m_masterFFWVel);
FOR i:=1 TO 3 DO
	m_cmdCartTwist[i] := m_masterFFVel[i];
	m_cmdCartTwist[i+3] := m_masterFFWVel[i];
END_FOR*)

// compute slave command pose in scope
vecSub(m_masterPose.m_pos, m_masterOriginPose.m_pos, masterMotionRange);

